         (*********************************************)
         (* parameter 3.7.3 *)
         (*********************************************)
         (
            ParameterName_as8    := 'POL Resistance Min',
            ParameterType_u8     := 0,
            attr1_u              := 0,
            attr2_u              := 3000,
            attr3_u              := 10,
            UnitCode_au8         := 18,
            Multiplier_s16       := 1,
            Divisor_s16          := 1,
            NumberOfDigits_u16   := 0,
            AccesslevelCode_u8   := 179,
            attr4_u              := 2,
            EEPROMAddress_s      := (Page_u8 := 3, IntIndex_u8 := 178)
         ),

         (*********************************************)
         (* parameter 3.7.4 *)
         (*********************************************)
         (
            ParameterName_as8    := 'POL Resistance Max',
            ParameterType_u8     := 0,
            attr1_u              := 0,
            attr2_u              := 3000,
            attr3_u              := 10,
            UnitCode_au8         := 18,
            Multiplier_s16       := 1,
            Divisor_s16          := 1,
            NumberOfDigits_u16   := 0,
            AccesslevelCode_u8   := 179,
            attr4_u              := 52,
            EEPROMAddress_s      := (Page_u8 := 3, IntIndex_u8 := 179)
         ),

         (*********************************************)
         (* parameter 3.7.5 *)
         (*********************************************)
         (
            ParameterName_as8    := 'POL Kp',
            ParameterType_u8     := 0,
            attr1_u              := 0,
            attr2_u              := 2000,
            attr3_u              := 50,
            UnitCode_au8         := 0,
            Multiplier_s16       := 1,
            Divisor_s16          := 1,
            NumberOfDigits_u16   := 0,
            AccesslevelCode_u8   := 179,
            attr4_u              := 250,
            EEPROMAddress_s      := (Page_u8 := 3, IntIndex_u8 := 180)
         ),

         (*********************************************)
         (* parameter 3.7.6 *)
         (*********************************************)
         (
            ParameterName_as8    := 'POL Ki',
            ParameterType_u8     := 0,
            attr1_u              := 0,
            attr2_u              := 500,
            attr3_u              := 50,
            UnitCode_au8         := 0,
            Multiplier_s16       := 1,
            Divisor_s16          := 1,
            NumberOfDigits_u16   := 0,
            AccesslevelCode_u8   := 179,
            attr4_u              := 250,
            EEPROMAddress_s      := (Page_u8 := 3, IntIndex_u8 := 181)
         ),

         (*********************************************)
         (* parameter 3.7.7 *)
         (*********************************************)
         (
         ),

         (*********************************************)
         (* parameter 3.7.8 *)
         (*********************************************)
         (
         )

      ),

      (*********************************************)
      (* parameter group 3.8 - up to 8 parameters can be defined here *)
      (*********************************************)
      (
         GroupName_as8   := 'DOH Configuration',

         Param_as        := 

         (*********************************************)
         (* parameter 3.8.1 *)
         (*********************************************)
         (
            ParameterName_as8    := 'DOH Debounce',
            ParameterType_u8     := 0,
            attr1_u              := 50,
            attr2_u              := 250,
            attr3_u              := 10,
            UnitCode_au8         := 4,
            Multiplier_s16       := 1,
            Divisor_s16          := 1,
            NumberOfDigits_u16   := 0,
            AccesslevelCode_u8   := 179,
            attr4_u              := 200,
            EEPROMAddress_s      := (Page_u8 := 3, IntIndex_u8 := 184)
         ),

         (*********************************************)
         (* parameter 3.8.2 *)
         (*********************************************)
         (
         ),

         (*********************************************)
         (* parameter 3.8.3 *)
         (*********************************************)
         (
            ParameterName_as8    := 'DOH Resistance Min',
            ParameterType_u8     := 0,
            attr1_u              := 0,
            attr2_u              := 3000,
            attr3_u              := 10,
            UnitCode_au8         := 18,
            Multiplier_s16       := 1,
            Divisor_s16          := 1,
            NumberOfDigits_u16   := 0,
            AccesslevelCode_u8   := 179,
            attr4_u              := 6,
            EEPROMAddress_s      := (Page_u8 := 3, IntIndex_u8 := 186)
         ),

         (*********************************************)
         (* parameter 3.8.4 *)
         (*********************************************)
         (
            ParameterName_as8    := 'DOH Resistance Max',
            ParameterType_u8     := 0,
            attr1_u              := 0,
            attr2_u              := 3000,
            attr3_u              := 10,
            UnitCode_au8         := 18,
            Multiplier_s16       := 1,
            Divisor_s16          := 1,
            NumberOfDigits_u16   := 0,
            AccesslevelCode_u8   := 179,
            attr4_u              := 44,
            EEPROMAddress_s      := (Page_u8 := 3, IntIndex_u8 := 187)
         ),

         (*********************************************)
         (* parameter 3.8.5 *)
         (*********************************************)
         (
         ),

         (*********************************************)
         (* parameter 3.8.6 *)
         (*********************************************)
         (
         ),

         (*********************************************)
         (* parameter 3.8.7 *)
         (*********************************************)
         (
         ),

         (*********************************************)
         (* parameter 3.8.8 *)
         (*********************************************)
         (
         )

      )

   ),

   (*********************************************)
   (* parameter menu 4 - up to 8 groups can be defined here *)
   (*********************************************)
   (
   ),

   (*********************************************)
   (* parameter menu 5 - up to 8 groups can be defined here *)
   (*********************************************)
   (
   );


(**)
END_VAR
(*********************************************)
(*  DON'T MAKE ANY CHANGES TO THIS PROGRAM!! *)
(*     FILE WAS AUTOMATICALLY GENERATED!!    *)
(*********************************************)

;
END_PROGRAM

(* POU 05_Basic_Calc/CHARCODE, ST *)
FUNCTION CHARCODE : BYTE
(* Функция получает код (char) для текстового символа *)
VAR_INPUT
	STR : STRING(1);
END_VAR
VAR
	PT : POINTER TO BYTE;
END_VAR
PT := ADR(STR);
CHARCODE := PT^;
END_FUNCTION

(* POU Uds/UdsSrvReadDataByIdServices/UdsGetProcessData, ST *)
PROGRAM UdsGetProcessData

VAR_INPUT
    did: UINT;
END_VAR

VAR
	startIndex: USINT := 1;
	groupNumber: USINT;
	requestedParameter: USINT;

	nonEmptyParametersCount: USINT;
	parameterCounter: USINT;
	numberOfParameters: USINT;
	parameterNameLength : USINT;

	tempCounter: USINT;
END_VAR
did := did - 16#2000;

groupNumber := UINT_TO_BYTE(SHR(did, 4));
groupNumber := groupNumber + 1;
requestedParameter := UINT_TO_BYTE(did) AND 16#0F;
requestedParameter := requestedParameter + 1;
Uds_s.UdsTx.data[1] := 0;

Uds_s.UdsTx.data[1] := Uds_s.UdsTx.data[1] + 1;
Uds_s.UdsTx.data[Uds_s.UdsTx.data[1] + 1 ] := Uds_s.UdsRx.data[2] + 16#40;

numberOfParameters := 8;

IF (LEN(ProcData.ProcessVarGroups_as[groupNumber].GroupName_as8) > 0) THEN
	IF (requestedParameter < 16#08) THEN
		startIndex := requestedParameter;
		numberOfParameters := startIndex;
	END_IF

	FOR parameterCounter := startIndex TO numberOfParameters DO
		parameterNameLength := INT_TO_USINT(LEN(ProcData.ProcessVarGroups_as[groupNumber].GroupName_as8));
		IF (parameterNameLength > 0) THEN
			nonEmptyParametersCount := nonEmptyParametersCount + 1;
		END_IF
	END_FOR

	Uds_s.UdsTx.data[1] := Uds_s.UdsTx.data[1] + 1;
	Uds_s.UdsTx.data[Uds_s.UdsTx.data[1] + 1] := nonEmptyParametersCount;

	FOR parameterCounter := startIndex TO numberOfParameters DO
		parameterNameLength := INT_TO_USINT(LEN(ProcData.ProcessVarGroups_as[groupNumber].GroupName_as8));
		IF (parameternameLength > 0) THEN
			Uds_s.UdsTx.data[1] := Uds_s.UdsTx.data[1] + 1;
			Uds_s.UdsTx.data[Uds_s.UdsTx.data[1] + 1] := parameterCounter - 1;

			IF (ProcData.ProcessVarGroups_as[groupNumber].ProcessVariable_as[parameterCounter].AccesslevelCode_u8 <= Uds_s.activeAccessLevel_u8) THEN
				FOR tempCounter := 1 TO parameterNameLength DO
					Uds_s.UdsTx.data[1] := Uds_s.UdsTx.data[1] + 1;
					Uds_s.UdsTx.data[Uds_s.UdsTx.data[1] + 1] := BYTE_TO_USINT(CHARCODE(MID(ProcData.ProcessVarGroups_as[groupNumber].ProcessVariable_as[parameterCounter].ProcessVarName_as8, 1, tempCounter)));
				END_FOR

				Uds_s.UdsTx.data[1] := Uds_s.UdsTx.data[1] + 1;
				Uds_s.UdsTx.data[Uds_s.UdsTx.data[1] + 1] := 0;

				Uds_s.UdsTx.data[1] := Uds_s.UdsTx.data[1] + 1;
				Uds_s.UdsTx.data[Uds_s.UdsTx.data[1] + 1] := INT_TO_USINT(SHR(ProcData.ProcessVarGroups_as[groupNumber].ProcessVariable_as[parameterCounter].Multiplier_s16, 8));
				Uds_s.UdsTx.data[1] := Uds_s.UdsTx.data[1] + 1;
				Uds_s.UdsTx.data[Uds_s.UdsTx.data[1] + 1] := INT_TO_USINT(ProcData.ProcessVarGroups_as[groupNumber].ProcessVariable_as[parameterCounter].Multiplier_s16);

				Uds_s.UdsTx.data[1] := Uds_s.UdsTx.data[1] + 1;
				Uds_s.UdsTx.data[Uds_s.UdsTx.data[1] + 1] := INT_TO_USINT(SHR(ProcData.ProcessVarGroups_as[groupNumber].ProcessVariable_as[parameterCounter].Divisor_s16, 8));
				Uds_s.UdsTx.data[1] := Uds_s.UdsTx.data[1] + 1;
				Uds_s.UdsTx.data[Uds_s.UdsTx.data[1] + 1] := INT_TO_USINT(ProcData.ProcessVarGroups_as[groupNumber].ProcessVariable_as[parameterCounter].Divisor_s16);

				Uds_s.UdsTx.data[1] := Uds_s.UdsTx.data[1] + 1;
				Uds_s.UdsTx.data[Uds_s.UdsTx.data[1] + 1] := ProcData.ProcessVarGroups_as[groupNumber].ProcessVariable_as[parameterCounter].ProcVarType_u8;

				Uds_s.UdsTx.data[1] := Uds_s.UdsTx.data[1] + 1;
				Uds_s.UdsTx.data[Uds_s.UdsTx.data[1] + 1] := UINT_TO_USINT(SHR(ProcData.ProcessVarGroups_as[groupNumber].ProcessVariable_as[parameterCounter].attr_u, 8));
				Uds_s.UdsTx.data[1] := Uds_s.UdsTx.data[1] + 1;
				Uds_s.UdsTx.data[Uds_s.UdsTx.data[1] + 1] := UINT_TO_USINT(ProcData.ProcessVarGroups_as[groupNumber].ProcessVariable_as[parameterCounter].attr_u);

				Uds_s.UdsTx.data[1] := Uds_s.UdsTx.data[1] + 1;
				Uds_s.UdsTx.data[Uds_s.UdsTx.data[1] + 1] := ProcData.ProcessVarGroups_as[groupNumber].ProcessVariable_as[parameterCounter].UnitCode_au8;

				Uds_s.UdsTx.data[1] := Uds_s.UdsTx.data[1] + 1;
				Uds_s.UdsTx.data[Uds_s.UdsTx.data[1] + 1] := ProcData.ProcessVarGroups_as[groupNumber].ProcessVariable_as[parameterCounter].AccesslevelCode_u8;

				IF (parameterCounter < numberOfParameters - 1 AND LEN(ProcData.ProcessVarGroups_as[groupNumber].ProcessVariable_as[parameterCounter + 1].ProcessVarName_as8) + 12 > (255 - Uds_s.UdsTx.data[1])) THEN
					EXIT;
				END_IF

			ELSE
				Uds_s.UdsTx.data[1] := Uds_s.UdsTx.data[1] + 1;
				Uds_s.UdsTx.data[Uds_s.UdsTx.data[1] + 1] := 0;
			END_IF
		END_IF
	END_FOR

	IF (parameterCounter = numberOfParameters + 1) THEN
		startIndex := 1;
	ELSE
		startIndex := parameterCounter + 1;
	END_IF
END_IF
Uds_s.UdsTx.dataSize := Uds_s.UdsTx.data[1];
END_PROGRAM

(* POU Autocode/ProcData, ST *)
PROGRAM ProcData
(*********************************************)
(*  DON'T MAKE ANY CHANGES TO THIS PROGRAM!! *)
(*     FILE WAS AUTOMATICALLY GENERATED!!    *)
(*********************************************)

VAR
END_VAR
VAR CONSTANT

(**)
(*********************************************)
nrProcMenus_u8          : USINT := 48;

(*********************************************)
(* Process Values Tree *)
(*********************************************)

ProcessVarGroups_as      : ARRAY [1..48] OF ProcessVariableGroup_ts := 

   (*********************************************)
   (* process values group 1 - up to 8 variables can be defined here *)
   (*********************************************)
   (
      GroupName_as8        := 'Group 1',

      ProcessVariable_as   := 

         (*********************************************)
      (* process value 1.1 *)
      (*********************************************)
      (
         ProcessVarName_as8   := 'Param_var',
         ProcVarType_u8       := 0,
         UnitCode_au8         := 1,
         Multiplier_s16       := 1,
         Divisor_s16          := 1,
         attr_u               := 0,
         AccesslevelCode_u8   := 129
      ),
         (*********************************************)
      (* process value 1.2 *)
      (*********************************************)
      (
         ProcessVarName_as8   := 'Param_var',
         ProcVarType_u8       := 0,
         UnitCode_au8         := 1,
         Multiplier_s16       := 1,
         Divisor_s16          := 1,
         attr_u               := 0,
         AccesslevelCode_u8   := 129
      ),
         (*********************************************)
      (* process value 1.3 *)
      (*********************************************)
      (
         ProcessVarName_as8   := 'Param_var',
         ProcVarType_u8       := 0,
         UnitCode_au8         := 1,
         Multiplier_s16       := 1,
         Divisor_s16          := 1,
         attr_u               := 0,
         AccesslevelCode_u8   := 129
      ),
         (*********************************************)
      (* process value 1.4 *)
      (*********************************************)
      (
         ProcessVarName_as8   := 'Param_var',
         ProcVarType_u8       := 0,
         UnitCode_au8         := 1,
         Multiplier_s16       := 1,
         Divisor_s16          := 1,
         attr_u               := 0,
         AccesslevelCode_u8   := 129
      ),
         (*********************************************)
      (* process value 1.5 *)
      (*********************************************)
      (
         ProcessVarName_as8   := 'Param_var',
         ProcVarType_u8       := 0,
         UnitCode_au8         := 0,
         Multiplier_s16       := 1,
         Divisor_s16          := 1,
         attr_u               := 0,
         AccesslevelCode_u8   := 129
      ),
         (*********************************************)
      (* process value 1.6 *)
      (*********************************************)
      (
         ProcessVarName_as8   := 'Param_var',
         ProcVarType_u8       := 0,
         UnitCode_au8         := 0,
         Multiplier_s16       := 1,
         Divisor_s16          := 1,
         attr_u               := 15,
         AccesslevelCode_u8   := 129
      ),
         (*********************************************)
      (* process value 1.7 *)
      (*********************************************)
      (
         ProcessVarName_as8   := 'Param_var',
         ProcVarType_u8       := 0,
         UnitCode_au8         := 0,
         Multiplier_s16       := 1,
         Divisor_s16          := 1,
         attr_u               := 8,
         AccesslevelCode_u8   := 129
      ),
         (*********************************************)
      (* process value 1.8 *)
      (*********************************************)
      (
         ProcessVarName_as8   := 'Param_var',
         ProcVarType_u8       := 0,
         UnitCode_au8         := 0,
         Multiplier_s16       := 1,
         Divisor_s16          := 1,
         attr_u               := 1000,
         AccesslevelCode_u8   := 129
      )
   ),

   (*********************************************)
   (* process values group 2 - up to 8 variables can be defined here *)
   (*********************************************)
   (
      GroupName_as8        := 'Group 2',

      ProcessVariable_as   := 

         (*********************************************)
      (* process value 2.1 *)
      (*********************************************)
      (
         ProcessVarName_as8   := 'Param_var',
         ProcVarType_u8       := 0,
         UnitCode_au8         := 1,
         Multiplier_s16       := 1,
         Divisor_s16          := 1,
         attr_u               := 0,
         AccesslevelCode_u8   := 129
      ),
         (*********************************************)
      (* process value 2.2 *)
      (*********************************************)
      (
         ProcessVarName_as8   := 'Param_var',
         ProcVarType_u8       := 0,
         UnitCode_au8         := 1,
         Multiplier_s16       := 1,
         Divisor_s16          := 1,
         attr_u               := 0,
         AccesslevelCode_u8   := 129
      ),
         (*********************************************)
      (* process value 2.3 *)
      (*********************************************)
      (
         ProcessVarName_as8   := 'Param_var',
         ProcVarType_u8       := 0,
         UnitCode_au8         := 1,
         Multiplier_s16       := 1,
         Divisor_s16          := 1,
         attr_u               := 0,
         AccesslevelCode_u8   := 129
      ),
         (*********************************************)
      (* process value 2.4 *)
      (*********************************************)
      (
         ProcessVarName_as8   := 'Param_var',
         ProcVarType_u8       := 0,
         UnitCode_au8         := 1,
         Multiplier_s16       := 1,
         Divisor_s16          := 1,
         attr_u               := 0,
         AccesslevelCode_u8   := 129
      ),
         (*********************************************)
      (* process value 2.5 *)
      (*********************************************)
      (
         ProcessVarName_as8   := 'Param_var',
         ProcVarType_u8       := 0,
         UnitCode_au8         := 1,
         Multiplier_s16       := 1,
         Divisor_s16          := 1,
         attr_u               := 0,
         AccesslevelCode_u8   := 129
      ),
         (*********************************************)
      (* process value 2.6 *)
      (*********************************************)
      (
         ProcessVarName_as8   := 'Param_var',
         ProcVarType_u8       := 0,
         UnitCode_au8         := 1,
         Multiplier_s16       := 1,
         Divisor_s16          := 1,
         attr_u               := 0,
         AccesslevelCode_u8   := 129
      ),
         (*********************************************)
      (* process value 2.7 *)
      (*********************************************)
      (
         ProcessVarName_as8   := 'Param_var',
         ProcVarType_u8       := 0,
         UnitCode_au8         := 1,
         Multiplier_s16       := 1,
         Divisor_s16          := 1,
         attr_u               := 0,
         AccesslevelCode_u8   := 129
      ),
         (*********************************************)
      (* process value 2.8 *)
      (*********************************************)
      (
         ProcessVarName_as8   := 'Param_var',
         ProcVarType_u8       := 0,
         UnitCode_au8         := 1,
         Multiplier_s16       := 1,
         Divisor_s16          := 1,
         attr_u               := 0,
         AccesslevelCode_u8   := 129
      )
   ),

   (*********************************************)
   (* process values group 3 - up to 8 variables can be defined here *)
   (*********************************************)
   (
      GroupName_as8        := 'Group 3',

      ProcessVariable_as   := 

         (*********************************************)
      (* process value 3.1 *)
      (*********************************************)
      (
         ProcessVarName_as8   := 'Param_var',
         ProcVarType_u8       := 0,
         UnitCode_au8         := 1,
         Multiplier_s16       := 1,
         Divisor_s16          := 1,
         attr_u               := 0,
         AccesslevelCode_u8   := 129
      ),
         (*********************************************)
      (* process value 3.2 *)
      (*********************************************)
      (
         ProcessVarName_as8   := 'Param_var',
         ProcVarType_u8       := 0,
         UnitCode_au8         := 1,
         Multiplier_s16       := 1,
         Divisor_s16          := 1,
         attr_u               := 0,
         AccesslevelCode_u8   := 129
      ),
         (*********************************************)
      (* process value 3.3 *)
      (*********************************************)
      (
         ProcessVarName_as8   := 'Param_var',
         ProcVarType_u8       := 0,
         UnitCode_au8         := 1,
         Multiplier_s16       := 1,
         Divisor_s16          := 1,
         attr_u               := 0,
         AccesslevelCode_u8   := 129
      ),
         (*********************************************)
      (* process value 3.4 *)
      (*********************************************)
      (
         ProcessVarName_as8   := 'Param_var',
         ProcVarType_u8       := 0,
         UnitCode_au8         := 1,
         Multiplier_s16       := 1,
         Divisor_s16          := 1,
         attr_u               := 0,
         AccesslevelCode_u8   := 129
      ),
         (*********************************************)
      (* process value 3.5 *)
      (*********************************************)
      (
         ProcessVarName_as8   := 'Param_var',
         ProcVarType_u8       := 0,
         UnitCode_au8         := 1,
         Multiplier_s16       := 1,
         Divisor_s16          := 1,
         attr_u               := 0,
         AccesslevelCode_u8   := 129
      ),
         (*********************************************)
      (* process value 3.6 *)
      (*********************************************)
      (
         ProcessVarName_as8   := 'Param_var',
         ProcVarType_u8       := 0,
         UnitCode_au8         := 1,
         Multiplier_s16       := 1,
         Divisor_s16          := 1,
         attr_u               := 0,
         AccesslevelCode_u8   := 129
      ),
         (*********************************************)
      (* process value 3.7 *)
      (*********************************************)
      (
         ProcessVarName_as8   := 'Param_var',
         ProcVarType_u8       := 0,
         UnitCode_au8         := 1,
         Multiplier_s16       := 1,
         Divisor_s16          := 1,
         attr_u               := 0,
         AccesslevelCode_u8   := 129
      ),
         (*********************************************)
      (* process value 3.8 *)
      (*********************************************)
      (
         ProcessVarName_as8   := 'Param_var',
         ProcVarType_u8       := 0,
         UnitCode_au8         := 1,
         Multiplier_s16       := 1,
         Divisor_s16          := 1,
         attr_u               := 0,
         AccesslevelCode_u8   := 129
      )
   ),

   (*********************************************)
   (* process values group 4 - up to 8 variables can be defined here *)
   (*********************************************)
   (
      GroupName_as8        := 'Group 4',

      ProcessVariable_as   := 

         (*********************************************)
      (* process value 4.1 *)
      (*********************************************)
      (
         ProcessVarName_as8   := 'Param_var',
         ProcVarType_u8       := 0,
         UnitCode_au8         := 1,
         Multiplier_s16       := 1,
         Divisor_s16          := 1,
         attr_u               := 0,
         AccesslevelCode_u8   := 129
      ),
         (*********************************************)
      (* process value 4.2 *)
      (*********************************************)
      (
         ProcessVarName_as8   := 'Param_var',
         ProcVarType_u8       := 0,
         UnitCode_au8         := 1,
         Multiplier_s16       := 1,
         Divisor_s16          := 1,
         attr_u               := 0,
         AccesslevelCode_u8   := 129
      ),
         (*********************************************)
      (* process value 4.3 *)
      (*********************************************)
      (
         ProcessVarName_as8   := 'Param_var',
         ProcVarType_u8       := 0,
         UnitCode_au8         := 1,
         Multiplier_s16       := 1,
         Divisor_s16          := 1,
         attr_u               := 0,
         AccesslevelCode_u8   := 129
      ),
         (*********************************************)
      (* process value 4.4 *)
      (*********************************************)
      (
         ProcessVarName_as8   := 'Param_var',
         ProcVarType_u8       := 0,
         UnitCode_au8         := 1,
         Multiplier_s16       := 1,
         Divisor_s16          := 1,
         attr_u               := 0,
         AccesslevelCode_u8   := 129
      ),
         (*********************************************)
      (* process value 4.5 *)
      (*********************************************)
      (
         ProcessVarName_as8   := 'Param_var',
         ProcVarType_u8       := 0,
         UnitCode_au8         := 1,
         Multiplier_s16       := 1,
         Divisor_s16          := 1,
         attr_u               := 0,
         AccesslevelCode_u8   := 129
      ),
         (*********************************************)
      (* process value 4.6 *)
      (*********************************************)
      (
         ProcessVarName_as8   := 'Param_var',
         ProcVarType_u8       := 0,
         UnitCode_au8         := 1,
         Multiplier_s16       := 1,
         Divisor_s16          := 1,
         attr_u               := 0,
         AccesslevelCode_u8   := 129
      ),
         (*********************************************)
      (* process value 4.7 *)
      (*********************************************)
      (
         ProcessVarName_as8   := 'Param_var',
         ProcVarType_u8       := 0,
         UnitCode_au8         := 1,
         Multiplier_s16       := 1,
         Divisor_s16          := 1,
         attr_u               := 0,
         AccesslevelCode_u8   := 129
      ),
         (*********************************************)
      (* process value 4.8 *)
      (*********************************************)
      (
      )
   ),

   (*********************************************)
   (* process values group 5 - up to 8 variables can be defined here *)
   (*********************************************)
   (
      GroupName_as8        := 'Group 5',

      ProcessVariable_as   := 

         (*********************************************)
      (* process value 5.1 *)
      (*********************************************)
      (
         ProcessVarName_as8   := 'Param_var',
         ProcVarType_u8       := 0,
         UnitCode_au8         := 1,
         Multiplier_s16       := 1,
         Divisor_s16          := 1,
         attr_u               := 0,
         AccesslevelCode_u8   := 129
      ),
         (*********************************************)
      (* process value 5.2 *)
      (*********************************************)
      (
         ProcessVarName_as8   := 'Param_var',
         ProcVarType_u8       := 0,
         UnitCode_au8         := 1,
         Multiplier_s16       := 1,
         Divisor_s16          := 1,
         attr_u               := 0,
         AccesslevelCode_u8   := 129
      ),
         (*********************************************)
      (* process value 5.3 *)
      (*********************************************)
      (
         ProcessVarName_as8   := 'Param_var',
         ProcVarType_u8       := 0,
         UnitCode_au8         := 1,
         Multiplier_s16       := 1,
         Divisor_s16          := 1,
         attr_u               := 0,
         AccesslevelCode_u8   := 129
      ),
         (*********************************************)
      (* process value 5.4 *)
      (*********************************************)
      (
         ProcessVarName_as8   := 'Param_var',
         ProcVarType_u8       := 0,
         UnitCode_au8         := 1,
         Multiplier_s16       := 1,
         Divisor_s16          := 1,
         attr_u               := 0,
         AccesslevelCode_u8   := 129
      ),
         (*********************************************)
      (* process value 5.5 *)
      (*********************************************)
      (
         ProcessVarName_as8   := 'Param_var',
         ProcVarType_u8       := 0,
         UnitCode_au8         := 1,
         Multiplier_s16       := 1,
         Divisor_s16          := 1,
         attr_u               := 0,
         AccesslevelCode_u8   := 129
      ),
         (*********************************************)
      (* process value 5.6 *)
      (*********************************************)
      (
         ProcessVarName_as8   := 'Param_var',
         ProcVarType_u8       := 0,
         UnitCode_au8         := 1,
         Multiplier_s16       := 1,
         Divisor_s16          := 1,
         attr_u               := 0,
         AccesslevelCode_u8   := 129
      ),
         (*********************************************)
      (* process value 5.7 *)
      (*********************************************)
      (
      ),
         (*********************************************)
      (* process value 5.8 *)
      (*********************************************)
      (
      )
   ),

   (*********************************************)
   (* process values group 6 - up to 8 variables can be defined here *)
   (*********************************************)
   (


   ),

   (*********************************************)
   (* process values group 7 - up to 8 variables can be defined here *)
   (*********************************************)
   (


   ),

   (*********************************************)
   (* process values group 8 - up to 8 variables can be defined here *)
   (*********************************************)
   (


   ),

   (*********************************************)
   (* process values group 9 - up to 8 variables can be defined here *)
   (*********************************************)
   (


   ),

   (*********************************************)
   (* process values group 10 - up to 8 variables can be defined here *)
   (*********************************************)
   (


   ),

   (*********************************************)
   (* process values group 11 - up to 8 variables can be defined here *)
   (*********************************************)
   (


   ),

   (*********************************************)
   (* process values group 12 - up to 8 variables can be defined here *)
   (*********************************************)
   (


   ),

   (*********************************************)
   (* process values group 13 - up to 8 variables can be defined here *)
   (*********************************************)
   (


   ),

   (*********************************************)
   (* process values group 14 - up to 8 variables can be defined here *)
   (*********************************************)
   (


   ),

   (*********************************************)
   (* process values group 15 - up to 8 variables can be defined here *)
   (*********************************************)
   (


   ),

   (*********************************************)
   (* process values group 16 - up to 8 variables can be defined here *)
   (*********************************************)
   (


   ),

   (*********************************************)
   (* process values group 17 - up to 8 variables can be defined here *)
   (*********************************************)
   (


   ),

   (*********************************************)
   (* process values group 18 - up to 8 variables can be defined here *)
   (*********************************************)
   (


   ),

   (*********************************************)
   (* process values group 19 - up to 8 variables can be defined here *)
   (*********************************************)
   (


   ),

   (*********************************************)
   (* process values group 20 - up to 8 variables can be defined here *)
   (*********************************************)
   (


   ),

   (*********************************************)
   (* process values group 21 - up to 8 variables can be defined here *)
   (*********************************************)
   (


   ),

   (*********************************************)
   (* process values group 22 - up to 8 variables can be defined here *)
   (*********************************************)
   (


   ),

   (*********************************************)
   (* process values group 23 - up to 8 variables can be defined here *)
   (*********************************************)
   (


   ),

   (*********************************************)
   (* process values group 24 - up to 8 variables can be defined here *)
   (*********************************************)
   (


   ),

   (*********************************************)
   (* process values group 25 - up to 8 variables can be defined here *)
   (*********************************************)
   (


   ),

   (*********************************************)
   (* process values group 26 - up to 8 variables can be defined here *)
   (*********************************************)
   (


   ),

   (*********************************************)
   (* process values group 27 - up to 8 variables can be defined here *)
   (*********************************************)
   (


   ),

   (*********************************************)
   (* process values group 28 - up to 8 variables can be defined here *)
   (*********************************************)
   (


   ),

   (*********************************************)
   (* process values group 29 - up to 8 variables can be defined here *)
   (*********************************************)
   (


   ),

   (*********************************************)
   (* process values group 30 - up to 8 variables can be defined here *)
   (*********************************************)
   (


   ),

   (*********************************************)
   (* process values group 31 - up to 8 variables can be defined here *)
   (*********************************************)
   (


   ),

   (*********************************************)
   (* process values group 32 - up to 8 variables can be defined here *)
   (*********************************************)
   (


   ),

   (*********************************************)
   (* process values group 33 - up to 8 variables can be defined here *)
   (*********************************************)
   (


   ),

   (*********************************************)
   (* process values group 34 - up to 8 variables can be defined here *)
   (*********************************************)
   (


   ),

   (*********************************************)
   (* process values group 35 - up to 8 variables can be defined here *)
   (*********************************************)
   (


   ),

   (*********************************************)
   (* process values group 36 - up to 8 variables can be defined here *)
   (*********************************************)
   (


   ),

   (*********************************************)
   (* process values group 37 - up to 8 variables can be defined here *)
   (*********************************************)
   (


   ),

   (*********************************************)
   (* process values group 38 - up to 8 variables can be defined here *)
   (*********************************************)
   (


   ),

   (*********************************************)
   (* process values group 39 - up to 8 variables can be defined here *)
   (*********************************************)
   (


   ),

   (*********************************************)
   (* process values group 40 - up to 8 variables can be defined here *)
   (*********************************************)
   (


   ),

   (*********************************************)
   (* process values group 41 - up to 8 variables can be defined here *)
   (*********************************************)
   (


   ),

   (*********************************************)
   (* process values group 42 - up to 8 variables can be defined here *)
   (*********************************************)
   (


   ),

   (*********************************************)
   (* process values group 43 - up to 8 variables can be defined here *)
   (*********************************************)
   (


   ),

   (*********************************************)
   (* process values group 44 - up to 8 variables can be defined here *)
   (*********************************************)
   (


   ),

   (*********************************************)
   (* process values group 45 - up to 8 variables can be defined here *)
   (*********************************************)
   (


   ),

   (*********************************************)
   (* process values group 46 - up to 8 variables can be defined here *)
   (*********************************************)
   (


   ),

   (*********************************************)
   (* process values group 47 - up to 8 variables can be defined here *)
   (*********************************************)
   (


   ),

   (*********************************************)
   (* process values group 48 - up to 8 variables can be defined here *)
   (*********************************************)
   (


   );


(**)
END_VAR
(*********************************************)
(*  DON'T MAKE ANY CHANGES TO THIS PROGRAM!! *)
(*     FILE WAS AUTOMATICALLY GENERATED!!    *)
(*********************************************)

;
END_PROGRAM

(* POU Uds/UdsSrvReadDataByIdServices/UdsGetParameterMenuNames, ST *)
PROGRAM UdsGetParameterMenuNames
VAR
	startIndex: USINT := 1;
	menuCounter: USINT;
	menuNameLength: USINT;

	nonEmptyMenuNamesCounter: USINT;
	tempCounter: USINT;
END_VAR
Uds_s.UdsTx.data[1] := 0;

Uds_s.UdsTx.data[1] := Uds_s.UdsTx.data[1] + 1;
Uds_s.UdsTx.data[Uds_s.UdsTx.data[1] + 1 ] := Uds_s.UdsRx.data[2] + 16#40;

FOR menuCounter := startIndex TO PrmData.nrPrmMenus_u8 DO
	menuNameLength := INT_TO_USINT(LEN(PrmData.ParameterMenus_as[menuCounter].MenuName_as8));
	IF (menuNameLength > 0) THEN
		nonEmptyMenuNamesCounter := nonEmptyMenuNamesCounter + 1;
	END_IF
END_FOR

Uds_s.UdsTx.data[1] := Uds_s.UdsTx.data[1] + 1;
Uds_s.UdsTx.data[Uds_s.UdsTx.data[1] + 1 ] := nonEmptyMenuNamesCounter;

FOR menuCounter := startIndex TO PrmData.nrPrmMenus_u8 DO
	menuNameLength := INT_TO_USINT(LEN(PrmData.ParameterMenus_as[menuCounter].MenuName_as8));
	IF (menuNameLength > 0) THEN
		Uds_s.UdsTx.data[1] := Uds_s.UdsTx.data[1] + 1;
		Uds_s.UdsTx.data[Uds_s.UdsTx.data[1] + 1] := menuCounter - 1;

		FOR tempCounter := 1 TO menuNameLength DO
			Uds_s.UdsTx.data[1] := Uds_s.UdsTx.data[1] + 1;
			Uds_s.UdsTx.data[Uds_s.UdsTx.data[1] + 1] := BYTE_TO_USINT(CHARCODE(MID(PrmData.ParameterMenus_as[menuCounter].MenuName_as8, 1, tempCounter)));
		END_FOR

		Uds_s.UdsTx.data[1] := Uds_s.UdsTx.data[1] + 1;
		Uds_s.UdsTx.data[Uds_s.UdsTx.data[1] + 1] := 0;

		IF (menuCounter < PrmData.nrPrmMenus_u8 - 1 AND LEN(PrmData.ParameterMenus_as[menuCounter + 1].MenuName_as8) + 3 > 255 - Uds_s.UdsTx.data[1]) THEN
			EXIT;
		END_IF
	END_IF
END_FOR
IF (menuCounter = PrmData.nrPrmMenus_u8 + 1) THEN
	startIndex := 1;
ELSE
	startIndex := menuCounter + 1;
END_IF
Uds_s.UdsTx.dataSize := Uds_s.UdsTx.data[1];
END_PROGRAM

(* POU Uds/UdsSrvReadDataByIdServices/UdsGetParameterSubMenuNames, ST *)
PROGRAM UdsGetParameterSubMenuNames

VAR_INPUT
    did: UINT;
END_VAR

VAR
	startIndex: USINT := 1;

	menuNumber: USINT;
	numberOfSubmenuNames: USINT := 8;
	subMenuCounter: USINT;
	nonEmptySubMenuNamesCounter: USINT;
	subMenuNameLength: USINT;

	tempCounter: USINT;
END_VAR
did := did - 16#2201;
menuNumber := UINT_TO_USINT(did);

Uds_s.UdsTx.data[1] := 0;
Uds_s.UdsTx.data[1] := Uds_s.UdsTx.data[1] + 1;
Uds_s.UdsTx.data[Uds_s.UdsTx.data[1] + 1 ] := Uds_s.UdsRx.data[2] + 16#40;

IF (LEN(PrmData.ParameterMenus_as[menuNumber].MenuName_as8) > 0) THEN
	FOR subMenuCounter := startIndex TO numberOfSubmenuNames DO
		subMenuNameLength := INT_TO_USINT(LEN(PrmData.ParameterMenus_as[menuNumber].ParameterGroup_as[subMenuCounter].GroupName_as8));
		IF (subMenuNameLength > 0) THEN
			nonEmptySubMenuNamesCounter := nonEmptySubMenuNamesCounter + 1;
		END_IF
	END_FOR

	Uds_s.UdsTx.data[1] := Uds_s.UdsTx.data[1] + 1;
	Uds_s.UdsTx.data[Uds_s.UdsTx.data[1] + 1 ] := nonEmptySubMenuNamesCounter;

	FOR subMenuCounter := startIndex TO numberOfSubmenuNames DO
		subMenuNameLength := INT_TO_USINT(LEN(PrmData.ParameterMenus_as[menuNumber].ParameterGroup_as[subMenuCounter].GroupName_as8));
		IF (subMenuNameLength > 0) THEN
			Uds_s.UdsTx.data[1] := Uds_s.UdsTx.data[1] + 1;
			Uds_s.UdsTx.data[Uds_s.UdsTx.data[1] + 1 ] := subMenuCounter;

			FOR tempCounter := 1 TO subMenuNameLength DO
				Uds_s.UdsTx.data[1] := Uds_s.UdsTx.data[1] + 1;
				Uds_s.UdsTx.data[Uds_s.UdsTx.data[1] + 1] := BYTE_TO_USINT(CHARCODE(MID(PrmData.ParameterMenus_as[menuNumber].ParameterGroup_as[subMenuCounter].GroupName_as8, 1, tempCounter)));
			END_FOR

			Uds_s.UdsTx.data[1] := Uds_s.UdsTx.data[1] + 1;
			Uds_s.UdsTx.data[Uds_s.UdsTx.data[1] + 1 ] := 0;

			IF (subMenuCounter < numberOfSubmenuNames - 1 AND LEN(PrmData.ParameterMenus_as[menuNumber].ParameterGroup_as[subMenuCounter + 1].GroupName_as8) + 3 > 255 - Uds_s.UdsTx.data[1]) THEN
				EXIT;
			END_IF
		END_IF
	END_FOR
	IF (subMenuCounter = numberOfSubmenuNames + 1) THEN
		startIndex := 1;
	ELSE
		startIndex := subMenuCounter + 1;
	END_IF
END_IF
Uds_s.UdsTx.dataSize := Uds_s.UdsTx.data[1];
END_PROGRAM

(* POU Uds/UdsSrvReadDataByIdServices/UdsGetProcessGroupNames, ST *)
PROGRAM UdsGetProcessGroupNames
VAR
    groupCounter : USINT;
    startIndex : USINT := 1;
    tempCounter : USINT;
    groupNameLength : USINT;
	nonEmptyGroupNamesCounter: USINT;
END_VAR
Uds_s.UdsTx.data[1] := Uds_s.UdsTx.data[1] + 1;
Uds_s.UdsTx.data[Uds_s.UdsTx.data[1] + 1 ] := Uds_s.UdsRx.data[2] + 16#40;

FOR groupCounter := startIndex TO ProcData.nrProcMenus_u8 DO
	groupNameLength := INT_TO_USINT(LEN(ProcData.ProcessVarGroups_as[groupCounter].GroupName_as8));
	IF (groupNameLength > 0) THEN
		nonEmptyGroupNamesCounter := nonEmptyGroupNamesCounter + 1;
	END_IF
END_FOR

Uds_s.UdsTx.data[1] := Uds_s.UdsTx.data[1] + 1;
Uds_s.UdsTx.data[Uds_s.UdsTx.data[1] + 1 ] := nonEmptyGroupNamesCounter;

FOR groupCounter := startIndex TO ProcData.nrProcMenus_u8 DO
    groupNameLength := INT_TO_USINT(LEN(ProcData.ProcessVarGroups_as[groupCounter].GroupName_as8));
    IF groupNameLength > 0 THEN
        Uds_s.UdsTx.data[1] := Uds_s.UdsTx.data[1] + 1;
        Uds_s.UdsTx.data[Uds_s.UdsTx.data[1] + 1] := groupCounter - 1;


        FOR tempCounter := 1 TO groupNameLength DO
            Uds_s.UdsTx.data[1] := Uds_s.UdsTx.data[1] + 1;
            Uds_s.UdsTx.data[Uds_s.UdsTx.data[1] + 1] := BYTE_TO_USINT(CHARCODE(MID(ProcData.ProcessVarGroups_as[groupCounter].GroupName_as8, 1, tempCounter)));
        END_FOR

        Uds_s.UdsTx.data[1] := Uds_s.UdsTx.data[1] + 1;
        Uds_s.UdsTx.data[Uds_s.UdsTx.data[1] + 1] := 0;
        IF (groupCounter < ProcData.nrProcMenus_u8 - 1 AND LEN(ProcData.ProcessVarGroups_as[groupCounter].GroupName_as8) + 3 > 255 - Uds_s.UdsTx.data[1]) THEN
            EXIT;
        END_IF
    END_IF
END_FOR
IF (groupCounter = ProcData.nrProcMenus_u8 + 1) THEN
    startIndex := 1;
ELSE
    startIndex := groupCounter + 1;
END_IF
Uds_s.UdsTx.dataSize := Uds_s.UdsTx.data[1];
END_PROGRAM

(* POU Uds/UdsSrvReadDataByIdServices/UdsGetUnitCodes, ST *)
PROGRAM UdsGetUnitCodes
VAR
    startIndex_u16 : USINT := 1;
    unitCodeCounter : USINT;
    tempCounter : USINT;
    unitCodeLength : USINT;
END_VAR
Uds_s.UdsTx.data[1] := 0;

Uds_s.UdsTx.data[1] := Uds_s.UdsTx.data[1] + 1;
Uds_s.UdsTx.data[Uds_s.UdsTx.data[1] + 1 ] := Uds_s.UdsRx.data[2] + 16#40;

Uds_s.UdsTx.data[1] := Uds_s.UdsTx.data[1] + 1;
Uds_s.UdsTx.data[Uds_s.UdsTx.data[1] + 1 ] := UnitCodes.nrUnitCodes_u8;

FOR unitCodeCounter := startIndex_u16 TO UnitCodes.nrUnitCodes_u8 DO
    Uds_s.UdsTx.data[1] := Uds_s.UdsTx.data[1] + 1;
    Uds_s.UdsTx.data[Uds_s.UdsTx.data[1] + 1] := unitCodeCounter - 1;
    unitCodeLength := INT_TO_USINT(LEN(UnitCodes.UnitCodes_cau8[unitCodeCounter]));
    FOR tempCounter := 1 TO unitCodeLength DO
        Uds_s.UdsTx.data[1] := Uds_s.UdsTx.data[1] + 1;
        Uds_s.UdsTx.data[Uds_s.UdsTx.data[1] + 1] := BYTE_TO_USINT(CHARCODE(MID(UnitCodes.UnitCodes_cau8[unitCodeCounter], 1, tempCounter)));
    END_FOR
    Uds_s.UdsTx.data[1] := Uds_s.UdsTx.data[1] + 1;
    Uds_s.UdsTx.data[Uds_s.UdsTx.data[1] + 1] := 0;

    IF (unitCodeCounter < UnitCodes.nrUnitCodes_u8 AND LEN(UnitCodes.UnitCodes_cau8[unitCodeCounter + 1]) + 3 > (255 - Uds_s.UdsTx.data[1])) THEN
        EXIT;
    END_IF
END_FOR

IF (unitCodeCounter = UnitCodes.nrUnitCodes_u8) THEN
    startIndex_u16 := 1;
ELSE
    startIndex_u16 := unitCodeCounter + 1;
END_IF
Uds_s.UdsTx.dataSize := Uds_s.UdsTx.data[1];
END_PROGRAM

(* POU Autocode/UnitCodes, ST *)
PROGRAM UnitCodes
(*********************************************)
(*  DON'T MAKE ANY CHANGES TO THIS PROGRAM!! *)
(*     FILE WAS AUTOMATICALLY GENERATED!!    *)
(*********************************************)

VAR
END_VAR
VAR CONSTANT

(**)
(*********************************************)
nrUnitCodes_u8      : USINT := 18;

(*********************************************)
(* Unit Codes Array *)

UnitCodes_cau8      : ARRAY [1..18] OF STRING(8) := 
   '%',
   'rpm',
   'hrs',
   'ms',
   'ccm',
   'mA',
   'bar',
   'mbar',
   'Deg C',
   'min',
   's',
   'km/h',
   'Nm',
   'deg °',
   '% / mA',
   '% / mV',
   'uA / mV',
   'Ohm';


(**)
END_VAR
(*********************************************)
(*  DON'T MAKE ANY CHANGES TO THIS PROGRAM!! *)
(*     FILE WAS AUTOMATICALLY GENERATED!!    *)
(*********************************************)

;
END_PROGRAM

(* POU Uds/UdsSrvReadDataByIdServices/UdsGetListDescriptions, ST *)
PROGRAM UdsGetListDescriptions
VAR
	listEntriesCounter: UINT;
	numberOfEntries: UINT;
	nonEmptyListDescriptionsCounter: UINT;
	listEntryLength: USINT;

	startIndex: UINT := 1;
	tempCounter: USINT;
END_VAR
Uds_s.UdsTx.data[1] := 0;

Uds_s.UdsTx.data[1] := Uds_s.UdsTx.data[1] + 1;
Uds_s.UdsTx.data[Uds_s.UdsTx.data[1] + 1 ] := Uds_s.UdsRx.data[2] + 16#40;

numberOfEntries := Lists.nrLists_u8 * 10;

FOR listEntriesCounter := startIndex TO numberOfEntries DO
	listEntryLength := INT_TO_USINT(LEN(Lists.ParaLists_as[listEntriesCounter / 10 + 1][listEntriesCounter MOD 10]));
	IF (listEntryLength > 0) THEN
		nonEmptyListDescriptionsCounter := nonEmptyListDescriptionsCounter + 1;
	END_IF
END_FOR

Uds_s.UdsTx.data[1] := Uds_s.UdsTx.data[1] + 1;
Uds_s.UdsTx.data[Uds_s.UdsTx.data[1] + 1 ] := UINT_TO_USINT(SHR(nonEmptyListDescriptionsCounter, 8));

Uds_s.UdsTx.data[1] := Uds_s.UdsTx.data[1] + 1;
Uds_s.UdsTx.data[Uds_s.UdsTx.data[1] + 1 ] := UINT_TO_USINT(nonEmptyListDescriptionsCounter);

Uds_s.UdsTx.data[1] := Uds_s.UdsTx.data[1] + 1;
Uds_s.UdsTx.data[Uds_s.UdsTx.data[1] + 1 ] := 10;

FOR listEntriesCounter := startIndex TO numberOfEntries DO
	listEntryLength := INT_TO_USINT(LEN(Lists.ParaLists_as[listEntriesCounter / 10 + 1][listEntriesCounter MOD 10]));
	IF (listEntryLength > 0) THEN
		Uds_s.UdsTx.data[1] := Uds_s.UdsTx.data[1] + 1;
		Uds_s.UdsTx.data[Uds_s.UdsTx.data[1] + 1 ] := UINT_TO_USINT(SHR(listEntriesCounter, 8));

		Uds_s.UdsTx.data[1] := Uds_s.UdsTx.data[1] + 1;
		Uds_s.UdsTx.data[Uds_s.UdsTx.data[1] + 1 ] := UINT_TO_USINT(listEntriesCounter);

		FOR tempCounter := 1 TO listEntryLength DO
			Uds_s.UdsTx.data[1] := Uds_s.UdsTx.data[1] + 1;
			Uds_s.UdsTx.data[Uds_s.UdsTx.data[1] + 1] := BYTE_TO_USINT(CHARCODE(MID(Lists.ParaLists_as[listEntriesCounter / 10 + 1][listEntriesCounter MOD 10], 1, tempCounter)));
		END_FOR

		Uds_s.UdsTx.data[1] := Uds_s.UdsTx.data[1] + 1;
		Uds_s.UdsTx.data[Uds_s.UdsTx.data[1] + 1] := 0;

		IF (listEntriesCounter <  numberOfEntries - 1 AND LEN(Lists.ParaLists_as[(listEntriesCounter + 1) / 10 + 1][(listEntriesCounter + 1) MOD 10]) > (255 - Uds_s.UdsTx.data[1])) THEN
			EXIT;
		END_IF
	END_IF
END_FOR

IF (listEntriesCounter = numberOfEntries + 1) THEN
	startIndex := 1;
ELSE
	startIndex := listEntriesCounter + 1;
END_IF

Uds_s.UdsTx.dataSize := Uds_s.UdsTx.data[1];
END_PROGRAM

(* POU Autocode/Lists, ST *)
PROGRAM Lists
(*********************************************)
(*  DON'T MAKE ANY CHANGES TO THIS PROGRAM!! *)
(*     FILE WAS AUTOMATICALLY GENERATED!!    *)
(*********************************************)

VAR
END_VAR
VAR CONSTANT

(**)
(*********************************************)
nrLists_u8      : USINT := 4;

(*********************************************)
(* Lists Tree*)

ParaLists_as      : ARRAY [1..4] OF ARRAY[1..10] OF STRING(32) := 
      'Not Active',
      'Active',
      '',
      '',
      '',
      '',
      '',
      '',
      '',
      '',
      'PWM',
      'PWM Current control',
      '',
      '',
      '',
      '',
      '',
      '',
      '',
      '',
      'PWM',
      'AOV',
      '',
      '',
      '',
      '',
      '',
      '',
      '',
      '',
      'AOC',
      'AOV',
      '',
      '',
      '',
      '',
      '',
      '',
      '',
      ''
;

(**)
END_VAR
(*********************************************)
(*  DON'T MAKE ANY CHANGES TO THIS PROGRAM!! *)
(*     FILE WAS AUTOMATICALLY GENERATED!!    *)
(*********************************************)

;
END_PROGRAM

(* POU Uds/UdsSrvReadDataByIdServices/UdsGetErrors, ST *)
PROGRAM UdsGetErrors
VAR_INPUT
    errorType: USINT;
END_VAR
VAR
    numErr : USINT;
    errorData : ARRAY[1..50] OF ErrorData_ts;
    errorCounter : USINT;
    startIndex : USINT := 1;
    tempCounter : USINT;
    errorListCounter : USINT;
    errorsEnum : applError_e;
END_VAR
Uds_s.UdsTx.data[1] := Uds_s.UdsTx.data[1] + 1;
Uds_s.UdsTx.data[Uds_s.UdsTx.data[1] + 1 ] := Uds_s.UdsRx.data[2] + 16#40;

IF (errorType = 0) THEN
    numErr := UINT_TO_USINT(sys_getSavedErrors(ADR(errorData[1]), 0, 50));
ELSIF (errorType = 1) THEN
    numErr := UINT_TO_USINT(sys_getActiveErrors(ADR(errorData[1]), 0, 50));
(*ELSE
    (*7F*)*)
END_IF

FOR errorCounter := startIndex TO numErr DO
    IF errorData[errorCounter].Code_u16 = 0 THEN
        EXIT;
    END_IF
    Uds_s.UdsTx.data[1] := Uds_s.UdsTx.data[1] + 1;
    Uds_s.UdsTx.data[Uds_s.UdsTx.data[1] + 1] := UINT_TO_USINT(SHR(errorData[errorCounter].Code_u16, 8));
    Uds_s.UdsTx.data[1] := Uds_s.UdsTx.data[1] + 1;
    Uds_s.UdsTx.data[Uds_s.UdsTx.data[1] + 1] := UINT_TO_USINT(errorData[errorCounter].Code_u16);
    Uds_s.UdsTx.data[1] := Uds_s.UdsTx.data[1] + 1;
    Uds_s.UdsTx.data[Uds_s.UdsTx.data[1] + 1] := errorData[errorCounter].Param_u8;
    Uds_s.UdsTx.data[1] := Uds_s.UdsTx.data[1] + 1;
    Uds_s.UdsTx.data[Uds_s.UdsTx.data[1] + 1] := errorData[errorCounter].Occurrence_u8;
    Uds_s.UdsTx.data[1] := Uds_s.UdsTx.data[1] + 1;
    Uds_s.UdsTx.data[Uds_s.UdsTx.data[1] + 1] := UDINT_TO_USINT(SHR(errorData[errorCounter].Timestamp_u32, 24));
    Uds_s.UdsTx.data[1] := Uds_s.UdsTx.data[1] + 1;
    Uds_s.UdsTx.data[Uds_s.UdsTx.data[1] + 1] := UDINT_TO_USINT(SHR(errorData[errorCounter].Timestamp_u32, 16));
    Uds_s.UdsTx.data[1] := Uds_s.UdsTx.data[1] + 1;
    Uds_s.UdsTx.data[Uds_s.UdsTx.data[1] + 1] := UDINT_TO_USINT(SHR(errorData[errorCounter].Timestamp_u32, 8));
    Uds_s.UdsTx.data[1] := Uds_s.UdsTx.data[1] + 1;
    Uds_s.UdsTx.data[Uds_s.UdsTx.data[1] + 1] := UDINT_TO_USINT(errorData[errorCounter].Timestamp_u32);

    FOR errorListCounter := 0 TO ErrorsList.nrErrors_u8 DO
        IF ErrorsList.ApplError_as[errorListCounter].Code_u16 = errorData[errorCounter].Code_u16 THEN
            FOR tempCounter := 0 TO INT_TO_USINT(LEN(ErrorsList.ApplError_as[errorListCounter].Description_as8)) DO
                Uds_s.UdsTx.data[1] := Uds_s.UdsTx.data[1] + 1;
                Uds_s.UdsTx.data[Uds_s.UdsTx.data[1] + 1] := BYTE_TO_USINT(CHARCODE(MID(ErrorsList.ApplError_as[errorListCounter].Description_as8, 1, tempCounter)));
            END_FOR
        END_IF
    END_FOR
END_FOR
IF (errorCounter = numErr + 1) THEN
    startIndex := 1;
ELSE
    startIndex := errorCounter + 1;
END_IF
Uds_s.UdsTx.dataSize := Uds_s.UdsTx.data[1];
END_PROGRAM

(* POU Autocode/ErrorsList, ST *)
PROGRAM ErrorsList
(*********************************************)
(*  DON'T MAKE ANY CHANGES TO THIS ENUMS!!   *)
(*     FILE WAS AUTOMATICALLY GENERATED!!    *)
(*********************************************)
VAR
END_VAR
VAR CONSTANT

(**)
(*********************************************)

(* Errors Tree *)
(*********************************************)
nrErrors_u8          : USINT := 21;

(*********************************************)
ApplError_as      : ARRAY [1..21] OF ApplErrorNew_ts := 

   (
      Code_u16 := 16#8000,
      Description_as8 := 'FIRST_CODE'
   ),
   (
      Code_u16 := 16#8001,
      Description_as8 := 'CAN_DIAG'
   ),
   (
      Code_u16 := 16#8036,
      Description_as8 := 'PWRON_SUPPLY_VB_LOW'
   ),
   (
      Code_u16 := 16#8037,
      Description_as8 := 'PWRON_SUPPLY_VSS'
   ),
   (
      Code_u16 := 16#8038,
      Description_as8 := 'PWRON_HWMONITOR_1'
   ),
   (
      Code_u16 := 16#8039,
      Description_as8 := 'PWRON_STARTCONDITION_1'
   ),
   (
      Code_u16 := 16#8040,
      Description_as8 := 'PWRON_ENGINE_SPEED'
   ),
   (
      Code_u16 := 16#8041,
      Description_as8 := 'PWRON_HWMONITOR_2'
   ),
   (
      Code_u16 := 16#8042,
      Description_as8 := 'PWRON_STARTCONDITION_2'
   ),
   (
      Code_u16 := 16#8043,
      Description_as8 := 'PWRON_SAFOUT_CABLE_BRAKE'
   ),
   (
      Code_u16 := 16#8044,
      Description_as8 := 'PWRON_SAFOUT_SHORT_CIRCUIT'
   ),
   (
      Code_u16 := 16#8045,
      Description_as8 := 'PWRON_POWERSWITCH_1'
   ),
   (
      Code_u16 := 16#8046,
      Description_as8 := 'PWRON_POWERSUPPLY'
   ),
   (
      Code_u16 := 16#8047,
      Description_as8 := 'PWRON_POWERSWITCH_2'
   ),
   (
      Code_u16 := 16#8048,
      Description_as8 := 'PWRON_REVERSE_POWER'
   ),
   (
      Code_u16 := 16#8049,
      Description_as8 := 'PWRON_EMERGENCY_STOP'
   ),
   (
      Code_u16 := 16#8031,
      Description_as8 := 'SUPPLY_VB_HIGH'
   ),
   (
      Code_u16 := 16#8032,
      Description_as8 := 'SUPPLY_VB_LOW'
   ),
   (
      Code_u16 := 16#8033,
      Description_as8 := 'SUPPLY_VSS1'
   ),
   (
      Code_u16 := 16#8034,
      Description_as8 := 'SUPPLY_VSS2'
   ),
   (
      Code_u16 := 16#8099,
      Description_as8 := 'LAST_CODE'
   )
(**)
;
END_VAR
(*********************************************)
(*  DON'T MAKE ANY CHANGES TO THIS PROGRAM!! *)
(*     FILE WAS AUTOMATICALLY GENERATED!!    *)
(*********************************************)

;
END_PROGRAM

(* POU Uds/UdsSrvReadDataByIdServices/UdsDidAcsPrm, ST *)
PROGRAM UdsDidAcsPrm
VAR_INPUT
	did: UINT;
   flgWrDid: USINT;
END_VAR
VAR
	menuNumber:USINT;
	subMenuNumber: USINT;
	parameterNumber: USINT;
	rawVal: UINT;
END_VAR
(* TODO
Запись: проверка на другие размеры передаваемого значения (1 байт, размер = 4)
*)
menuNumber := UINT_TO_BYTE(SHR(did, 7)) AND 16#3F;
menuNumber := menuNumber + 1;
subMenuNumber := UINT_TO_BYTE(SHR(did, 4)) AND 16#07;
subMenuNumber := subMenuNumber + 1;
parameterNumber := UINT_TO_BYTE(did) AND 16#0F;
parameterNumber := parameterNumber + 1;

IF (menuNumber <= PrmData.nrPrmMenus_u8) THEN

Uds_s.UdsTx.data[1] := 0;

Uds_s.UdsTx.data[1] := Uds_s.UdsTx.data[1] + 1;
Uds_s.UdsTx.data[Uds_s.UdsTx.data[1] + 1 ] := Uds_s.UdsRx.data[2] + 16#40;

IF (flgWrDid = 0) THEN (*read access*)
	rawVal := ree_getValue(PrmData.ParameterMenus_as[menuNumber].ParameterGroup_as[subMenuNumber].Param_as[parameterNumber].EEPROMAddress_s.Page_u8,
									PrmData.ParameterMenus_as[menuNumber].ParameterGroup_as[subMenuNumber].Param_as[parameterNumber].EEPROMAddress_s.IntIndex_u8);
	Uds_s.UdsTx.data[1] := Uds_s.UdsTx.data[1] + 1;
	Uds_s.UdsTx.data[Uds_s.UdsTx.data[1] + 1 ] := UINT_TO_USINT(SHR(did, 8));
	Uds_s.UdsTx.data[1] := Uds_s.UdsTx.data[1] + 1;
	Uds_s.UdsTx.data[Uds_s.UdsTx.data[1] + 1 ] := UINT_TO_USINT(did);

ELSE (*write access*)
	IF Uds_s.UdsRx.dataSize = 5 THEN (*1 - sid; 2,3 - did; 4,5 - value*)
		rawVal := USINT_TO_UINT(SHL(Uds_s.UdsRx.data[4], 8));
		rawVal := rawVal + Uds_s.UdsRx.data[5];
		IF (rawVal > PrmData.ParameterMenus_as[menuNumber].ParameterGroup_as[subMenuNumber].Param_as[parameterNumber].attr1_u AND
				rawVal < PrmData.ParameterMenus_as[menuNumber].ParameterGroup_as[subMenuNumber].Param_as[parameterNumber].attr2_u) THEN
			ree_setValue(PrmData.ParameterMenus_as[menuNumber].ParameterGroup_as[subMenuNumber].Param_as[parameterNumber].EEPROMAddress_s.Page_u8,
								PrmData.ParameterMenus_as[menuNumber].ParameterGroup_as[subMenuNumber].Param_as[parameterNumber].EEPROMAddress_s.IntIndex_u8,
								rawVal);
		END_IF
	END_IF
END_IF
Uds_s.UdsTx.dataSize := Uds_s.UdsTx.data[1];

END_IF
END_PROGRAM

(* POU Uds/UdsSrvReadDataByIdServices/UdsDidAcsProcVal, ST *)
PROGRAM UdsDidAcsProcVal
VAR_INPUT
	did : UINT;
END_VAR
VAR
END_VAR
;
END_PROGRAM

(* POU Uds/UdsSrvWriteDataById, ST *)
PROGRAM UdsSrvWriteDataById
VAR
	didus : UINT;
END_VAR
IF (Uds_s.UdsRx.dataSize > 0 AND Uds_s.UdsRx.data[1] > 0) THEN
	didus := Uds_s.UdsRx.data[3];
	didus := SHL(didus, 8);
	didus := didus + Uds_s.UdsRx.data[4];

	UdsDidAcsPrm(did := didus, flgWrDid := 1);
END_IF
END_PROGRAM

(* POU Uds/UdsSrvTesterPresent, ST *)
PROGRAM UdsSrvTesterPresent
VAR

END_VAR
IF(Uds_s.UdsRx.dataSize = 2) THEN
	Uds_s.UdsTx.data[1] := 0;
	
	Uds_s.UdsTx.data[1] := Uds_s.UdsTx.data[1] + 1;
	Uds_s.UdsTx.data[Uds_s.UdsTx.data[1] + 1 ] := Uds_s.UdsRx.data[2] + 16#40;

	Uds_s.UdsTx.data[1] := Uds_s.UdsTx.data[1] + 1;
	Uds_s.UdsTx.data[Uds_s.UdsTx.data[1] + 1 ] := 16#00;
	
	Uds_s.UdsTx.dataSize := Uds_s.UdsTx.data[1];
END_IF
END_PROGRAM

(* POU Autocode/Callback_update_appl_param, ST *)
(*************************************************************************************
BRIEF: read the whole parameters from the EEPROM
*************************************************************************************
 (c) Copyright by BOSCH REXROTH AG, all rights reserved 
*************************************************************************************
VERSION INFORMATION
	V1.0 	Vitaly Lewitan, DC-MA/SMC
- Call Autocode parameter assignment programm
- Update (or Init) function block parameters

REVISION HISTORY:
	V1.0 	Vitaly Lewitan, DC-MA/SMC
 - 23/03-2012 Initial Version
**************************************************************************************)
PROGRAM Callback_update_appl_param

VAR
   eep:  ARRAY [0..1280] OF INT;
END_VAR
Callback_diag_getPara();
(* Get_Aggregate_param(); *)
END_PROGRAM

(* POU Autocode/Callback_diag_getPara, ST *)
PROGRAM Callback_diag_getPara
VAR
   eep:  ARRAY [0..1280] OF INT;
END_VAR
(*********************************************)
(*  DON'T MAKE ANY CHANGES TO THIS PROGRAM!! *)
(*     FILE WAS AUTOMATICALLY GENERATED!!    *)
(*********************************************)

(* get EEPROM pages 0..4 *)
ree_getArray( PAGE0, 0, ADR(eep[0]),    256 );
ree_getArray( PAGE1, 0, ADR(eep[256]),  256 );
ree_getArray( PAGE2, 0, ADR(eep[512]),  256 );
ree_getArray( PAGE3, 0, ADR(eep[768]),  256 );
ree_getArray( PAGE4, 0, ADR(eep[1024]), 256 );


(* Menu 1 *)

(* Basic *)
para_s.number_1_1_1_s16 := eep[EEP_number_1_1_1_e];
para_s.Input_to_Output_Mode_s16 := eep[EEP_Input_to_Output_Mode_e];
para_s.test_par_new_s16 := eep[EEP_test_par_new_e];
para_s.test_params_s16 := eep[EEP_test_params_e];
para_s.test_par2_s16 := eep[EEP_test_par2_e];

(* Test Type *)
para_s.Trimming_type_s16 := eep[EEP_Trimming_type_e];
para_s.Analog_type_s16 := eep[EEP_Analog_type_e];
para_s.Curve_Type_s16 := eep[EEP_Curve_Type_e];
para_s.Function_Type_s16 := eep[EEP_Function_Type_e];
para_s.Percent_Type_s16 := eep[EEP_Percent_Type_e];
para_s.Ramp_Type_s16 := eep[EEP_Ramp_Type_e];
para_s.Switch_Type_s16 := eep[EEP_Switch_Type_e];
para_s.List_Type_s16 := eep[EEP_List_Type_e];

(* Test Number *)
para_s.number_1_3_1_s16 := eep[EEP_number_1_3_1_e];
para_s.number_1_3_2_s16 := eep[EEP_number_1_3_2_e];
para_s.number_1_3_3_s16 := eep[EEP_number_1_3_3_e];
para_s.number_1_3_4_s16 := eep[EEP_number_1_3_4_e];
para_s.number_1_3_5_s16 := eep[EEP_number_1_3_5_e];
para_s.number_1_3_6_s16 := eep[EEP_number_1_3_6_e];
para_s.number_1_3_7_s16 := eep[EEP_number_1_3_7_e];
para_s.number_1_3_8_s16 := eep[EEP_number_1_3_8_e];


(* Menu 2 *)

(* Output Cfg 1-8 *)
para_s.Out_Cfg_01_s16 := eep[EEP_Out_Cfg_01_e];
para_s.Out_Cfg_02_s16 := eep[EEP_Out_Cfg_02_e];
para_s.Out_Cfg_03_s16 := eep[EEP_Out_Cfg_03_e];
para_s.Out_Cfg_04_s16 := eep[EEP_Out_Cfg_04_e];
para_s.Out_Cfg_05_s16 := eep[EEP_Out_Cfg_05_e];
para_s.Out_Cfg_06_s16 := eep[EEP_Out_Cfg_06_e];
para_s.Out_Cfg_07_s16 := eep[EEP_Out_Cfg_07_e];
para_s.Out_Cfg_08_s16 := eep[EEP_Out_Cfg_08_e];

(* Output Cfg 9-16 *)
para_s.Out_Cfg_09_s16 := eep[EEP_Out_Cfg_09_e];
para_s.Out_Cfg_10_s16 := eep[EEP_Out_Cfg_10_e];
para_s.Out_Cfg_11_s16 := eep[EEP_Out_Cfg_11_e];
para_s.Out_Cfg_12_s16 := eep[EEP_Out_Cfg_12_e];
para_s.Out_Cfg_13_s16 := eep[EEP_Out_Cfg_13_e];
para_s.Out_Cfg_14_s16 := eep[EEP_Out_Cfg_14_e];
para_s.Out_Cfg_15_s16 := eep[EEP_Out_Cfg_15_e];
para_s.Out_Cfg_16_s16 := eep[EEP_Out_Cfg_16_e];

(* Output Cfg 17-24 *)
para_s.Out_Cfg_17_s16 := eep[EEP_Out_Cfg_17_e];
para_s.Out_Cfg_18_s16 := eep[EEP_Out_Cfg_18_e];
para_s.Out_Cfg_19_s16 := eep[EEP_Out_Cfg_19_e];
para_s.Out_Cfg_20_s16 := eep[EEP_Out_Cfg_20_e];
para_s.Out_Cfg_21_s16 := eep[EEP_Out_Cfg_21_e];
para_s.Out_Cfg_22_s16 := eep[EEP_Out_Cfg_22_e];
para_s.Out_Cfg_23_s16 := eep[EEP_Out_Cfg_23_e];
para_s.Out_Cfg_24_s16 := eep[EEP_Out_Cfg_24_e];

(* Output Cfg 25-32 *)
para_s.Out_Cfg_25_s16 := eep[EEP_Out_Cfg_25_e];
para_s.Out_Cfg_26_s16 := eep[EEP_Out_Cfg_26_e];
para_s.Out_Cfg_27_s16 := eep[EEP_Out_Cfg_27_e];
para_s.Out_Cfg_28_s16 := eep[EEP_Out_Cfg_28_e];
para_s.Out_Cfg_29_s16 := eep[EEP_Out_Cfg_29_e];
para_s.Out_Cfg_30_s16 := eep[EEP_Out_Cfg_30_e];
para_s.Out_Cfg_31_s16 := eep[EEP_Out_Cfg_31_e];
para_s.Out_Cfg_32_s16 := eep[EEP_Out_Cfg_32_e];

(* Output Cfg 33-40 *)
para_s.Out_Cfg_33_s16 := eep[EEP_Out_Cfg_33_e];
para_s.Out_Cfg_34_s16 := eep[EEP_Out_Cfg_34_e];
para_s.Out_Cfg_35_s16 := eep[EEP_Out_Cfg_35_e];
para_s.Out_Cfg_36_s16 := eep[EEP_Out_Cfg_36_e];
para_s.Out_Cfg_37_s16 := eep[EEP_Out_Cfg_37_e];
para_s.Out_Cfg_38_s16 := eep[EEP_Out_Cfg_38_e];
para_s.Out_Cfg_39_s16 := eep[EEP_Out_Cfg_39_e];
para_s.Out_Cfg_40_s16 := eep[EEP_Out_Cfg_40_e];

(* Output Cfg 41-47 *)
para_s.Out_Cfg_41_s16 := eep[EEP_Out_Cfg_41_e];
para_s.Out_Cfg_42_s16 := eep[EEP_Out_Cfg_42_e];
para_s.Out_Cfg_43_s16 := eep[EEP_Out_Cfg_43_e];
para_s.Out_Cfg_44_s16 := eep[EEP_Out_Cfg_44_e];
para_s.Out_Cfg_45_s16 := eep[EEP_Out_Cfg_45_e];
para_s.Out_Cfg_46_s16 := eep[EEP_Out_Cfg_46_e];
para_s.Out_Cfg_47_s16 := eep[EEP_Out_Cfg_47_e];

(* AOV Configuration *)
para_s.AOV_Debounce_s16 := eep[EEP_AOV_Debounce_e];
para_s.AOV_Freq_s16 := eep[EEP_AOV_Freq_e];
para_s.AOV_Res_Min_s16 := eep[EEP_AOV_Res_Min_e];
para_s.AOV_Res_Max_s16 := eep[EEP_AOV_Res_Max_e];
para_s.AOV_Kp_s16 := eep[EEP_AOV_Kp_e];
para_s.AOV_Ki_s16 := eep[EEP_AOV_Ki_e];

(* AOC Configuration *)
para_s.AOC_Debounce_s16 := eep[EEP_AOC_Debounce_e];
para_s.AOC_Freq_s16 := eep[EEP_AOC_Freq_e];
para_s.AOC_Res_Min_s16 := eep[EEP_AOC_Res_Min_e];
para_s.AOC_Res_Max_s16 := eep[EEP_AOC_Res_Max_e];
para_s.AOC_Kp_s16 := eep[EEP_AOC_Kp_e];
para_s.AOC_Ki_s16 := eep[EEP_AOC_Ki_e];


(* Menu 3 *)

(* Output Value 1-8 *)
para_s.Out_Val_01_s16 := eep[EEP_Out_Val_01_e];
para_s.Out_Val_02_s16 := eep[EEP_Out_Val_02_e];
para_s.Out_Val_03_s16 := eep[EEP_Out_Val_03_e];
para_s.Out_Val_04_s16 := eep[EEP_Out_Val_04_e];
para_s.Out_Val_05_s16 := eep[EEP_Out_Val_05_e];
para_s.Out_Val_06_s16 := eep[EEP_Out_Val_06_e];
para_s.Out_Val_07_s16 := eep[EEP_Out_Val_07_e];
para_s.Out_Val_08_s16 := eep[EEP_Out_Val_08_e];

(* Output Value 9-16 *)
para_s.Out_Val_09_s16 := eep[EEP_Out_Val_09_e];
para_s.Out_Val_10_s16 := eep[EEP_Out_Val_10_e];
para_s.Out_Val_11_s16 := eep[EEP_Out_Val_11_e];
para_s.Out_Val_12_s16 := eep[EEP_Out_Val_12_e];
para_s.Out_Val_13_s16 := eep[EEP_Out_Val_13_e];
para_s.Out_Val_14_s16 := eep[EEP_Out_Val_14_e];
para_s.Out_Val_15_s16 := eep[EEP_Out_Val_15_e];
para_s.Out_Val_16_s16 := eep[EEP_Out_Val_16_e];

(* Output Value 17-36 *)
para_s.Out_Val_17_s16 := eep[EEP_Out_Val_17_e];
para_s.Out_Val_18_s16 := eep[EEP_Out_Val_18_e];
para_s.Out_Val_33_s16 := eep[EEP_Out_Val_33_e];
para_s.Out_Val_34_s16 := eep[EEP_Out_Val_34_e];
para_s.Out_Val_35_s16 := eep[EEP_Out_Val_35_e];
para_s.Out_Val_36_s16 := eep[EEP_Out_Val_36_e];

(* Output Value 37-44 *)
para_s.Out_Val_37_s16 := eep[EEP_Out_Val_37_e];
para_s.Out_Val_38_s16 := eep[EEP_Out_Val_38_e];
para_s.Out_Val_39_s16 := eep[EEP_Out_Val_39_e];
para_s.Out_Val_40_s16 := eep[EEP_Out_Val_40_e];
para_s.Out_Val_41_s16 := eep[EEP_Out_Val_41_e];
para_s.Out_Val_42_s16 := eep[EEP_Out_Val_42_e];
para_s.Out_Val_43_s16 := eep[EEP_Out_Val_43_e];
para_s.Out_Val_44_s16 := eep[EEP_Out_Val_44_e];

(* Output Value 45-47 *)
para_s.Out_Val_45_s16 := eep[EEP_Out_Val_45_e];
para_s.Out_Val_46_s16 := eep[EEP_Out_Val_46_e];
para_s.Out_Val_47_s16 := eep[EEP_Out_Val_47_e];

(* POH Configuration *)
para_s.POH_Debounce_s16 := eep[EEP_POH_Debounce_e];
para_s.POH_Res_Min_s16 := eep[EEP_POH_Res_Min_e];
para_s.POH_Res_Max_s16 := eep[EEP_POH_Res_Max_e];
para_s.POH_Kp_s16 := eep[EEP_POH_Kp_e];
para_s.POH_Ki_s16 := eep[EEP_POH_Ki_e];

(* POL Configuration *)
para_s.POL_Debounce_s16 := eep[EEP_POL_Debounce_e];
para_s.POL_Res_Min_s16 := eep[EEP_POL_Res_Min_e];
para_s.POL_Res_Max_s16 := eep[EEP_POL_Res_Max_e];
para_s.POL_Kp_s16 := eep[EEP_POL_Kp_e];
para_s.POL_Ki_s16 := eep[EEP_POL_Ki_e];

(* DOH Configuration *)
para_s.DOH_Debounce_s16 := eep[EEP_DOH_Debounce_e];
para_s.DOH_Res_Min_s16 := eep[EEP_DOH_Res_Min_e];
para_s.DOH_Res_Max_s16 := eep[EEP_DOH_Res_Max_e];
END_PROGRAM

(* POU SwInfo, ST *)
PROGRAM SwInfo
VAR

	SwInfo_lenString_DU32	: INT := 255;
	Eep_sizePage_16bit_D		: INT := 256;

	SwInfo_strSep_DAS8		: STRING := ' |-| \n\r';
	SwInfo_dataString_as8	: STRING(255);

	idx_u16						: INT := 1;

	flgCompRes_u8				: BOOL := FALSE;

	SwInfo_dataEepromRd_as16 : ARRAY[1..256] OF INT := 0;
	SwInfo_dataEepromWr_as16 : ARRAY[1..256] OF INT := 0;

	Ecu_nrEepPageEcuInfo_D	: INT := 32;
END_VAR
(* copy constant SW Name string to target *)
SwInfo_dataString_as8 := 'Software Git Commit Hash: ';
SwInfo_dataString_as8 := CONCAT(SwInfo_dataString_as8, SW_Version.SW_Git_Hash_as8);
SwInfo_dataString_as8 := CONCAT(SwInfo_dataString_as8, ';');


(* switch byte order in string *)
(* Switch byte order of characters in string to prepare string for display in BODAS service *)
FOR idx_u16 := 1 TO SwInfo_lenString_DU32 BY 1 DO
	IF (idx_u16 MOD 2 = 0) THEN
		(* odd byte position *)
		SwInfo_dataEepromWr_as16[idx_u16/2] := WORD_TO_INT(INT_TO_WORD(SwInfo_dataEepromWr_as16[idx_u16/2]) OR (BYTE_TO_WORD(CHARCODE(MID(SwInfo_dataString_as8, 1, idx_u16)))  AND 16#00FF));
	ELSE
		(* even byte position *)
		SwInfo_dataEepromWr_as16[idx_u16/2 + 1] :=  WORD_TO_INT(SHL(BYTE_TO_WORD(CHARCODE(MID(SwInfo_dataString_as8, 1, idx_u16))),8) AND 16#FF00);
	END_IF
END_FOR

(* read current content of EEPROM RAM mirror page containing ECU information *)
ree_getArray(Ecu_nrEepPageEcuInfo_D, 0, ADR(SwInfo_dataEepromRd_as16[1]), Eep_sizePage_16bit_D);

(* create index for array comparison *)
idx_u16 := 1;

(* create flag holding array comparison result *)
flgCompRes_u8 := FALSE;
(* -------------------------------------------------------------------------------------------- *)

(* compare actual content with intended content *)
WHILE ((idx_u16 < Eep_sizePage_16bit_D) AND (NOT flgCompRes_u8)) DO
	IF (SwInfo_dataEepromRd_as16[idx_u16] <> SwInfo_dataEepromWr_as16[idx_u16]) THEN
		flgCompRes_u8 := TRUE;
	END_IF
	idx_u16 := idx_u16 + 1;
END_WHILE

IF (flgCompRes_u8) THEN
	ee_saveArray(Ecu_nrEepPageEcuInfo_D, 0, ADR(SwInfo_dataEepromWr_as16[1]), Eep_sizePage_16bit_D);
END_IF
END_PROGRAM

(* POU 10_Inputs/General Parameters/Get_System_Info, ST *)
PROGRAM Get_System_Info
VAR
	stSupplyVP1_b8			: BOOL;	(*state of the supply VP1*)
	stSupplyVP2_b8			: BOOL;	(*state of the supply VP2*)

	tiSysRunTime_s32		: DINT;	(*duration of the task*)
	etaSysTaskLoad_s16	: INT;	(*load of the main task*)

	stSysEMCY_b8			: BOOL; (*State of the emergency switch*)
	stSysINH_b8				: BOOL;	(*State of INH (pin228)*)

	PCB_temp_s16			: INT;  (*temperature of the RC*)

	error_u16				: UINT;	(* ECU info error *)
	EcuInfo_s				: EcuInfo_ts;
   errors_u16				: ARRAY [1..19] OF UINT;
   BufferAPPL_au8			: ARRAY [1..32] OF USINT;
   BufferSB_au8			: ARRAY [1..6] OF USINT;
   BufferCB_au8			: ARRAY [1..6] OF USINT;
   BufferAPI_au8			: ARRAY [1..1024] OF USINT;
   BufferAPs_au8			: ARRAY [1..19] OF ARRAY [1..16] OF USINT;
   copiedBytes_u16		: ARRAY [1..19] OF UINT;
END_VAR
(********************************************************************************************)
(******************** Checkt:INH / EMCY state  **********************************************)
(********************************************************************************************)
(*check the state OF 'INH': excepted value: OFF*)
stSysINH_b8		:= USINT_TO_BOOL(sys_getINH());
stSysEMCY_b8	:= emcy_getStatus( );
(******************************************************************************)
(******************** Read Supply Voltage  ************************************)
(******************************************************************************)
(* check VP switches *)
stSupplyVP1_b8		:= sys_getVP( VP_1 );			(* State of the supply VP1 *)
stSupplyVP2_b8		:= sys_getVP( VP_2 );			(* State of the supply VP2 *)
(******************************************************************************)
(******************** Read Task data  *****************************************)
(******************************************************************************)
tiSysRunTime_s32 		:= sys_getTaskRunTime( PLC_PRG.MAIN_Task_Handle_u8, PTIME_AVERAGE_INCL );
etaSysTaskLoad_s16 	:= sys_getTaskLoad(PTIME_AVERAGE_INCL);
(******************************************************************************)
(******************** Reads the PCB (Printed circuit board) temperature in °C**)
(******************************************************************************)
PCB_temp_s16 := sys_getHwTemp(AIT_HW_1);

(* Get information of the electronic circuit unit (ECU) *)
error_u16 := sys_getEcuInfo(ADR(EcuInfo_s));

(*
errors_u16[1] 	:= sys_getVersion(VERSION_SW_PART_APPL_DU8 					, ADR(BufferAPPL_au8[1]), 	32,	ADR(copiedBytes_u16[1]));
errors_u16[2] 	:= sys_getVersion(VERSION_SW_PART_SB_DU8						, ADR(BufferSB_au8[1]), 	6, 	ADR(copiedBytes_u16[2]));
errors_u16[3] 	:= sys_getVersion(VERSION_SW_PART_CB_DU8						, ADR(BufferCB_au8[1]), 	6, 	ADR(copiedBytes_u16[3]));
errors_u16[4] 	:= sys_getVersion(VERSION_SW_PART_API_ALL_DU8 				, ADR(BufferAPI_au8[1]), 	1024,	ADR(copiedBytes_u16[4]));
errors_u16[5] 	:= sys_getVersion(VERSION_SW_PART_API_BASIC_DU8 			, ADR(BufferAPs_au8[5]), 	16,	ADR(copiedBytes_u16[5]));
errors_u16[6] 	:= sys_getVersion(VERSION_SW_PART_API_SRC_RC_BASIC_DU8 	, ADR(BufferAPs_au8[6]), 	16,	ADR(copiedBytes_u16[6]));
errors_u16[7] 	:= sys_getVersion(VERSION_SW_PART_API_EEPROM_DU8 			, ADR(BufferAPs_au8[7]), 	16,	ADR(copiedBytes_u16[7]));
errors_u16[8] 	:= sys_getVersion(VERSION_SW_PART_API_DIAG_DU8 				, ADR(BufferAPs_au8[8]), 	16,	ADR(copiedBytes_u16[8]));
errors_u16[9] 	:= sys_getVersion(VERSION_SW_PART_API_INEXT_DU8 			, ADR(BufferAPs_au8[9]), 	16,	ADR(copiedBytes_u16[9]));
errors_u16[10] := sys_getVersion(VERSION_SW_PART_API_STM_DU8	 			, ADR(BufferAPs_au8[10]), 	16,	ADR(copiedBytes_u16[10]));
errors_u16[11] := sys_getVersion(VERSION_SW_PART_API_CANOPEN_DU8 			, ADR(BufferAPs_au8[11]), 	16,	ADR(copiedBytes_u16[11]));
errors_u16[12] := sys_getVersion(VERSION_SW_PART_API_J1939_DU8 			, ADR(BufferAPs_au8[12]), 	16,	ADR(copiedBytes_u16[12]));
errors_u16[13] := sys_getVersion(VERSION_SW_PART_API_RTS_DU8	 			, ADR(BufferAPs_au8[13]), 	16,	ADR(copiedBytes_u16[13]));
errors_u16[14] := sys_getVersion(VERSION_SW_PART_API_CANOPEN_RCE_DU8		, ADR(BufferAPs_au8[14]), 	16,	ADR(copiedBytes_u16[14]));
errors_u16[15] := sys_getVersion(VERSION_SW_PART_API_UDS_DU8	 			, ADR(BufferAPs_au8[15]), 	16,	ADR(copiedBytes_u16[15]));
errors_u16[16] := sys_getVersion(VERSION_SW_PART_API_OUTEXT_DU8 			, ADR(BufferAPs_au8[16]), 	16,	ADR(copiedBytes_u16[16]));
errors_u16[17] := sys_getVersion(VERSION_SW_PART_API_ACOM_DU8	 			, ADR(BufferAPs_au8[17]), 	16,	ADR(copiedBytes_u16[17]));
errors_u16[18]	:= sys_getVersion(VERSION_SW_PART_API_RTM_DU8	 			, ADR(BufferAPs_au8[18]), 	16,	ADR(copiedBytes_u16[18]));
errors_u16[19]	:= sys_getVersion(VERSION_SW_PART_API_CCP_DU8	 			, ADR(BufferAPs_au8[19]), 	16,	ADR(copiedBytes_u16[19]));
*)
END_PROGRAM

(* POU 30_Outputs/out_Control, ST *)
PROGRAM out_Control
VAR
	out_19_state_b8	: BOOL;	(* Состояние выхода out_19 *)
	out_19_status_s	: out_ts;	(* Статус выхода out_19 *)
	out_19_on_b8		: BOOL;

	out_Brakes_status_s	: out_ts;	(* Статус выхода out_19 *)
	out_Brakes_on_b8		: BOOL;
END_VAR
VAR CONSTANT
	DOH_DUTYCYCLE_ON		: UINT	:= 10000;	(* Скважность, при которой дискретный выход активирован *)
END_VAR
IF para_s.Input_to_Output_Mode_s16 = DEACTIVATED THEN


	out_POH();
	out_DOH();
	out_AOV();
	out_POL();

IF PLC_PRG.EcuInfo_s.HwType_u16 <> PLC_PRG.HW_Type_RC12_10_30_u16 THEN
	out_getStatusxt(IO_Chnl.DOH_BRAKES, ADR(out_Brakes_status_s));
	out_Brakes_on_b8		:= out_Brakes_status_s.out_po_s.dc_u16 = DOH_DUTYCYCLE_ON;

	out(IO_Chnl.DOH_FLASHING_BEACON,	BOOL_TO_INT(out_Brakes_on_b8));							(* Выход маяка *)
END_IF

ELSE


;
END_IF
END_PROGRAM
ACTION out_AOV:
IF para_s.Out_Cfg_33_s16 = PWM_MODE THEN
	out (	OUT_33_POH,	para_s.Out_Val_33_s16);
ELSIF para_s.Out_Cfg_33_s16 = AOV_MODE THEN
	out (	OUT_33_AOV,	para_s.Out_Val_33_s16);
END_IF

IF para_s.Out_Cfg_34_s16 = PWM_MODE THEN
	out (	OUT_34_POH,	para_s.Out_Val_34_s16);
ELSIF para_s.Out_Cfg_34_s16 = AOV_MODE THEN
	out (	OUT_34_AOV,	para_s.Out_Val_34_s16);
END_IF

IF para_s.Out_Cfg_35_s16 = PWM_MODE THEN
	out (	OUT_35_POH,	para_s.Out_Val_35_s16);
ELSIF para_s.Out_Cfg_35_s16 = AOV_MODE THEN
	out (	OUT_35_AOV,	para_s.Out_Val_35_s16);
END_IF

IF para_s.Out_Cfg_36_s16 = PWM_MODE THEN
	out (	OUT_36_POH,	para_s.Out_Val_36_s16);
ELSIF para_s.Out_Cfg_36_s16 = AOV_MODE THEN
	out (	OUT_36_AOV,	para_s.Out_Val_36_s16);
END_IF

IF para_s.Out_Cfg_47_s16 = AOC_MODE THEN
	out (	OUT_47_AOC,	para_s.Out_Val_47_s16);
ELSIF para_s.Out_Cfg_47_s16 = AOV_MODE THEN
	out (	OUT_47_AOV,	para_s.Out_Val_47_s16);
END_IF
END_ACTION
ACTION out_DOH:
out(OUT_19_DOH, para_s.Out_Cfg_19_s16);
out(OUT_20_DOH, para_s.Out_Cfg_20_s16);
out(OUT_21_DOH, para_s.Out_Cfg_21_s16);
out(OUT_22_DOH, para_s.Out_Cfg_22_s16);
out(OUT_23_DOH, para_s.Out_Cfg_23_s16);
out(OUT_24_DOH, para_s.Out_Cfg_24_s16);
out(OUT_25_DOH, para_s.Out_Cfg_25_s16);
out(OUT_26_DOH, para_s.Out_Cfg_26_s16);
out(OUT_27_DOH, para_s.Out_Cfg_27_s16);
out(OUT_28_DOH, para_s.Out_Cfg_28_s16);
out(OUT_29_DOH, para_s.Out_Cfg_29_s16);
out(OUT_30_DOH, para_s.Out_Cfg_30_s16);
out(OUT_31_DOH, para_s.Out_Cfg_31_s16);
out(OUT_32_DOH, para_s.Out_Cfg_32_s16);
END_ACTION
ACTION out_POH:
(* Proportional output high side PWM *)

IF para_s.Out_Cfg_01_s16 = PWM_MODE THEN
	out (	OUT_1_POH,	para_s.Out_Val_01_s16);
ELSIF para_s.Out_Cfg_01_s16 = PWM_CURRENT_MODE THEN
	out (	OUT_1_POH_CL,	para_s.Out_Val_01_s16);
END_IF

IF para_s.Out_Cfg_02_s16 = PWM_MODE THEN
	out (	OUT_2_POH,	para_s.Out_Val_02_s16);
ELSIF para_s.Out_Cfg_01_s16 = PWM_CURRENT_MODE THEN
	out (	OUT_2_POH_CL,	para_s.Out_Val_02_s16);
END_IF

IF para_s.Out_Cfg_03_s16 = PWM_MODE THEN
	out (	OUT_3_POH,	para_s.Out_Val_03_s16);
ELSIF para_s.Out_Cfg_03_s16 = PWM_CURRENT_MODE THEN
	out (	OUT_3_POH_CL,	para_s.Out_Val_03_s16);
END_IF

IF para_s.Out_Cfg_04_s16 = PWM_MODE THEN
	out (	OUT_4_POH,	para_s.Out_Val_04_s16);
ELSIF para_s.Out_Cfg_04_s16 = PWM_CURRENT_MODE THEN
	out (	OUT_4_POH_CL,	para_s.Out_Val_04_s16);
END_IF

IF para_s.Out_Cfg_05_s16 = PWM_MODE THEN
	out (	OUT_5_POH,	para_s.Out_Val_05_s16);
ELSIF para_s.Out_Cfg_05_s16 = PWM_CURRENT_MODE THEN
	out (	OUT_5_POH_CL,	para_s.Out_Val_05_s16);
END_IF

IF para_s.Out_Cfg_06_s16 = PWM_MODE THEN
	out (	OUT_6_POH,	para_s.Out_Val_06_s16);
ELSIF para_s.Out_Cfg_06_s16 = PWM_CURRENT_MODE THEN
	out (	OUT_6_POH_CL,	para_s.Out_Val_06_s16);
END_IF

IF para_s.Out_Cfg_07_s16 = PWM_MODE THEN
	out (	OUT_7_POH,	para_s.Out_Val_07_s16);
ELSIF para_s.Out_Cfg_07_s16 = PWM_CURRENT_MODE THEN
	out (	OUT_7_POH_CL,	para_s.Out_Val_07_s16);
END_IF

IF para_s.Out_Cfg_08_s16 = PWM_MODE THEN
	out (	OUT_8_POH,	para_s.Out_Val_08_s16);
ELSIF para_s.Out_Cfg_08_s16 = PWM_CURRENT_MODE THEN
	out (	OUT_8_POH_CL,	para_s.Out_Val_08_s16);
END_IF

IF para_s.Out_Cfg_09_s16 = PWM_MODE THEN
	out (	OUT_9_POH,	para_s.Out_Val_09_s16);
ELSIF para_s.Out_Cfg_09_s16 = PWM_CURRENT_MODE THEN
	out (	OUT_9_POH_CL,	para_s.Out_Val_09_s16);
END_IF

IF para_s.Out_Cfg_10_s16 = PWM_MODE THEN
	out (	OUT_10_POH,	para_s.Out_Val_10_s16);
ELSIF para_s.Out_Cfg_10_s16 = PWM_CURRENT_MODE THEN
	out (	OUT_10_POH_CL,	para_s.Out_Val_10_s16);
END_IF

IF para_s.Out_Cfg_11_s16 = PWM_MODE THEN
	out (	OUT_11_POH,	para_s.Out_Val_11_s16);
ELSIF para_s.Out_Cfg_11_s16 = PWM_CURRENT_MODE THEN
	out (	OUT_11_POH_CL,	para_s.Out_Val_11_s16);
END_IF

IF para_s.Out_Cfg_12_s16 = PWM_MODE THEN
	out (	OUT_12_POH,	para_s.Out_Val_12_s16);
ELSIF para_s.Out_Cfg_12_s16 = PWM_CURRENT_MODE THEN
	out (	OUT_12_POH_CL,	para_s.Out_Val_12_s16);
END_IF

IF para_s.Out_Cfg_13_s16 = PWM_MODE THEN
	out (	OUT_13_POH,	para_s.Out_Val_13_s16);
ELSIF para_s.Out_Cfg_13_s16 = PWM_CURRENT_MODE THEN
	out (	OUT_13_POH_CL,	para_s.Out_Val_13_s16);
END_IF

IF para_s.Out_Cfg_14_s16 = PWM_MODE THEN
	out (	OUT_14_POH,	para_s.Out_Val_14_s16);
ELSIF para_s.Out_Cfg_14_s16 = PWM_CURRENT_MODE THEN
	out (	OUT_14_POH_CL,	para_s.Out_Val_14_s16);
END_IF

IF para_s.Out_Cfg_15_s16 = PWM_MODE THEN
	out (	OUT_15_POH,	para_s.Out_Val_15_s16);
ELSIF para_s.Out_Cfg_15_s16 = PWM_CURRENT_MODE THEN
	out (	OUT_15_POH_CL,	para_s.Out_Val_15_s16);
END_IF

IF para_s.Out_Cfg_16_s16 = PWM_MODE THEN
	out (	OUT_16_POH,	para_s.Out_Val_16_s16);
ELSIF para_s.Out_Cfg_16_s16 = PWM_CURRENT_MODE THEN
	out (	OUT_16_POH_CL,	para_s.Out_Val_16_s16);
END_IF

IF para_s.Out_Cfg_17_s16 = PWM_MODE THEN
	out (	OUT_17_POH,	para_s.Out_Val_17_s16);
ELSIF para_s.Out_Cfg_17_s16 = PWM_CURRENT_MODE THEN
	out (	OUT_17_POH_CL,	para_s.Out_Val_17_s16);
END_IF

IF para_s.Out_Cfg_18_s16 = PWM_MODE THEN
	out (	OUT_18_POH,	para_s.Out_Val_18_s16);
ELSIF para_s.Out_Cfg_18_s16 = PWM_CURRENT_MODE THEN
	out (	OUT_18_POH_CL,	para_s.Out_Val_18_s16);
END_IF
END_ACTION
ACTION out_POL:
(* Proportional output Low side PWM *)

IF para_s.Out_Cfg_37_s16 = PWM_MODE THEN
	out (	OUT_37_POL,	para_s.Out_Val_37_s16);
ELSIF para_s.Out_Cfg_37_s16 = PWM_CURRENT_MODE THEN
	out (	OUT_37_POL_CL,	para_s.Out_Val_37_s16);
END_IF

IF para_s.Out_Cfg_38_s16 = PWM_MODE THEN
	out (	OUT_38_POL,	para_s.Out_Val_38_s16);
ELSIF para_s.Out_Cfg_38_s16 = PWM_CURRENT_MODE THEN
	out (	OUT_38_POL_CL,	para_s.Out_Val_38_s16);
END_IF

IF para_s.Out_Cfg_39_s16 = PWM_MODE THEN
	out (	OUT_39_POL,	para_s.Out_Val_39_s16);
ELSIF para_s.Out_Cfg_39_s16 = PWM_CURRENT_MODE THEN
	out (	OUT_39_POL_CL,	para_s.Out_Val_39_s16);
END_IF

IF para_s.Out_Cfg_40_s16 = PWM_MODE THEN
	out (	OUT_40_POL,	para_s.Out_Val_40_s16);
ELSIF para_s.Out_Cfg_40_s16 = PWM_CURRENT_MODE THEN
	out (	OUT_40_POL_CL,	para_s.Out_Val_40_s16);
END_IF

IF para_s.Out_Cfg_41_s16 = PWM_MODE THEN
	out (	OUT_41_POL,	para_s.Out_Val_14_s16);
ELSIF para_s.Out_Cfg_14_s16 = PWM_CURRENT_MODE THEN
	out (	OUT_41_POL_CL,	para_s.Out_Val_41_s16);
END_IF

IF para_s.Out_Cfg_42_s16 = PWM_MODE THEN
	out (	OUT_42_POL,	para_s.Out_Val_42_s16);
ELSIF para_s.Out_Cfg_42_s16 = PWM_CURRENT_MODE THEN
	out (	OUT_42_POL_CL,	para_s.Out_Val_42_s16);
END_IF

IF para_s.Out_Cfg_43_s16 = PWM_MODE THEN
	out (	OUT_43_POL,	para_s.Out_Val_43_s16);
ELSIF para_s.Out_Cfg_43_s16 = PWM_CURRENT_MODE THEN
	out (	OUT_43_POL_CL,	para_s.Out_Val_43_s16);
END_IF

IF para_s.Out_Cfg_44_s16 = PWM_MODE THEN
	out (	OUT_44_POL,	para_s.Out_Val_44_s16);
ELSIF para_s.Out_Cfg_44_s16 = PWM_CURRENT_MODE THEN
	out (	OUT_44_POL_CL,	para_s.Out_Val_44_s16);
END_IF

IF para_s.Out_Cfg_45_s16 = PWM_MODE THEN
	out (	OUT_45_POL,	para_s.Out_Val_45_s16);
ELSIF para_s.Out_Cfg_45_s16 = PWM_CURRENT_MODE THEN
	out (	OUT_45_POL_CL,	para_s.Out_Val_45_s16);
END_IF

IF para_s.Out_Cfg_46_s16 = PWM_MODE THEN
	out (	OUT_46_POL,	para_s.Out_Val_46_s16);
ELSIF para_s.Out_Cfg_46_s16 = PWM_CURRENT_MODE THEN
	out (	OUT_46_POL_CL,	para_s.Out_Val_46_s16);
END_IF
END_ACTION

(* POU 30_Outputs/out_Current, ST *)
PROGRAM out_Current
VAR
END_VAR
(********************************************************************************)
(***** Получение актуальных значений токов PWM выходов **************************)
(********************************************************************************)

(* Test Code *)
output.iAct_Out_01_ma_s32			:= in( OUT_1_PIC );
output.iAct_Out_02_ma_s32			:= in( OUT_2_PIC );
output.iAct_Out_03_ma_s32			:= in( OUT_3_PIC );
output.iAct_Out_04_ma_s32			:= in( OUT_4_PIC );

(* code for test *)
output.iAct_Out_02_ma_s32			:= in( OUT_2_PIC );
output.iAct_Out_03_ma_s32			:= in( OUT_3_PIC );
output.iAct_Out_04_ma_s32			:= in( OUT_4_PIC );
output.iAct_Out_05_ma_s32			:= in( OUT_5_PIC );

output.iAct_Out_01_ma_s32			:= in( OUT_1_PIC );
output.iAct_Out_02_ma_s32			:= in( OUT_2_PIC );
output.iAct_Out_03_ma_s32			:= in( OUT_3_PIC );
output.iAct_Out_04_ma_s32			:= in( OUT_4_PIC );
output.iAct_Out_05_ma_s32			:= in( OUT_5_PIC );
output.iAct_Out_06_ma_s32			:= in( OUT_6_PIC );
output.iAct_Out_07_ma_s32			:= in( OUT_7_PIC );
output.iAct_Out_08_ma_s32			:= in( OUT_8_PIC );
output.iAct_Out_09_ma_s32			:= in( OUT_9_PIC );
output.iAct_Out_10_ma_s32			:= in( OUT_10_PIC);
output.iAct_Out_11_ma_s32			:= in( OUT_11_PIC);
output.iAct_Out_12_ma_s32			:= in( OUT_12_PIC);
output.iAct_Out_13_ma_s32			:= in( OUT_13_PIC);
output.iAct_Out_14_ma_s32			:= in( OUT_14_PIC);
output.iAct_Out_15_ma_s32			:= in( OUT_15_PIC);
output.iAct_Out_16_ma_s32			:= in( OUT_16_PIC);
output.iAct_Out_17_ma_s32			:= in( OUT_17_PIC);
output.iAct_Out_18_ma_s32			:= in( OUT_18_PIC);
output.iAct_Out_19_ma_s32			:= in( OUT_19_PIC);
output.iAct_Out_20_ma_s32			:= in( OUT_20_PIC);
output.iAct_Out_21_ma_s32			:= in( OUT_21_PIC);
output.iAct_Out_22_ma_s32			:= in( OUT_22_PIC);
output.iAct_Out_23_ma_s32			:= in( OUT_23_PIC);
output.iAct_Out_24_ma_s32			:= in( OUT_24_PIC);
output.iAct_Out_25_ma_s32			:= in( OUT_25_PIC);
output.iAct_Out_26_ma_s32			:= in( OUT_26_PIC);
output.iAct_Out_27_ma_s32			:= in( OUT_27_PIC);
output.iAct_Out_28_ma_s32			:= in( OUT_28_PIC);
output.iAct_Out_29_ma_s32			:= in( OUT_29_PIC);
output.iAct_Out_30_ma_s32			:= in( OUT_30_PIC);
output.iAct_Out_31_ma_s32			:= in( OUT_31_PIC);
output.iAct_Out_32_ma_s32			:= in( OUT_32_PIC);
output.iAct_Out_37_ma_s32			:= in( OUT_37_PIC);
output.iAct_Out_38_ma_s32			:= in( OUT_38_PIC);
output.iAct_Out_39_ma_s32			:= in( OUT_39_PIC);
output.iAct_Out_40_ma_s32			:= in( OUT_40_PIC);
output.iAct_Out_41_ma_s32			:= in( OUT_41_PIC);
output.iAct_Out_42_ma_s32			:= in( OUT_42_PIC);
output.iAct_Out_43_ma_s32			:= in( OUT_43_PIC);
output.iAct_Out_44_ma_s32			:= in( OUT_44_PIC);
output.iAct_Out_45_ma_s32			:= in( OUT_45_PIC);
output.iAct_Out_46_ma_s32			:= in( OUT_46_PIC);
END_PROGRAM

(* POU 30_Outputs/out_Status, ST *)
PROGRAM out_Status
VAR

	out_as: ARRAY [1..75] OF out_ts;	(* Structure with the extended output information *)

END_VAR
out_getStatusxt(OUT_1_POH,		ADR(out_as[1]));
out_getStatusxt(OUT_2_POH,		ADR(out_as[2]));
out_getStatusxt(OUT_3_POH, 	ADR(out_as[3]));
out_getStatusxt(OUT_4_POH, 	ADR(out_as[4]));
out_getStatusxt(OUT_5_POH, 	ADR(out_as[5]));
out_getStatusxt(OUT_6_POH, 	ADR(out_as[6]));
out_getStatusxt(OUT_7_POH, 	ADR(out_as[7]));
out_getStatusxt(OUT_8_POH, 	ADR(out_as[8]));
out_getStatusxt(OUT_9_POH, 	ADR(out_as[9]));
out_getStatusxt(OUT_10_POH, 	ADR(out_as[10]));
out_getStatusxt(OUT_11_POH, 	ADR(out_as[11]));
out_getStatusxt(OUT_12_POH, 	ADR(out_as[12]));
out_getStatusxt(OUT_13_POH, 	ADR(out_as[13]));
out_getStatusxt(OUT_14_POH,	ADR(out_as[14]));
out_getStatusxt(OUT_15_POH,	ADR(out_as[15]));
out_getStatusxt(OUT_16_POH, 	ADR(out_as[16]));
out_getStatusxt(OUT_17_POH,	ADR(out_as[17]));
out_getStatusxt(OUT_18_POH,	ADR(out_as[18]));
out_getStatusxt(OUT_19_DOH,	ADR(out_as[19]));
out_getStatusxt(OUT_20_DOH,	ADR(out_as[20]));
out_getStatusxt(OUT_21_DOH,	ADR(out_as[21]));
out_getStatusxt(OUT_22_DOH,	ADR(out_as[22]));
out_getStatusxt(OUT_23_DOH,	ADR(out_as[23]));
out_getStatusxt(OUT_24_DOH,	ADR(out_as[24]));
out_getStatusxt(OUT_25_DOH,	ADR(out_as[25]));
out_getStatusxt(OUT_26_DOH,	ADR(out_as[26]));
out_getStatusxt(OUT_27_DOH,	ADR(out_as[27]));
out_getStatusxt(OUT_28_DOH,	ADR(out_as[28]));
out_getStatusxt(OUT_29_DOH,	ADR(out_as[29]));
out_getStatusxt(OUT_30_DOH,	ADR(out_as[30]));
out_getStatusxt(OUT_31_DOH,	ADR(out_as[31]));
out_getStatusxt(OUT_32_DOH,	ADR(out_as[32]));
out_getStatusxt(OUT_33_POH,	ADR(out_as[33]));
out_getStatusxt(OUT_34_POH,	ADR(out_as[34]));
out_getStatusxt(OUT_35_POH,	ADR(out_as[35]));
out_getStatusxt(OUT_36_POH,	ADR(out_as[36]));
out_getStatusxt(OUT_37_POL,	ADR(out_as[37]));
out_getStatusxt(OUT_38_POL,	ADR(out_as[38]));
out_getStatusxt(OUT_39_POL,	ADR(out_as[39]));
out_getStatusxt(OUT_40_POL,	ADR(out_as[40]));
out_getStatusxt(OUT_41_POL,	ADR(out_as[41]));
out_getStatusxt(OUT_42_POL,	ADR(out_as[42]));
out_getStatusxt(OUT_43_POL,	ADR(out_as[43]));
out_getStatusxt(OUT_44_POL,	ADR(out_as[44]));
out_getStatusxt(OUT_45_POL,	ADR(out_as[45]));
out_getStatusxt(OUT_46_POL,	ADR(out_as[46]));
out_getStatusxt(OUT_47_AOV,	ADR(out_as[47]));

(* test code *)
out_getStatusxt(OUT_42_POL,	ADR(out_as[42]));
out_getStatusxt(OUT_43_POL,	ADR(out_as[43]));
out_getStatusxt(OUT_44_POL,	ADR(out_as[44]));
out_getStatusxt(OUT_45_POL,	ADR(out_as[45]));
out_getStatusxt(OUT_46_POL,	ADR(out_as[46]));
out_getStatusxt(OUT_47_AOV,	ADR(out_as[47]));
END_PROGRAM

(* POU 60_Error handling/Process Errors/proc_Err_DIG_outs, ST *)
PROGRAM proc_Err_DIG_outs
VAR

END_VAR
;
END_PROGRAM

(* POU 60_Error handling/Process Errors/proc_Err_Inputs, ST *)
PROGRAM proc_Err_Inputs
VAR

(*		Here we process errors from sensors, or HMI - which have to be calibrated at the beginning
		 = 0 no error, > 0 error
		Encoding of error bits:
			Bit 0x0000 = no error
			Bit 0x0004 = potentiometer slider < lower error threshold value (only if error threshold value >0)
			Bit 0x0008 = potentiometer slider > upper error threshold value
			Bit 0x0020 = potentiometer slider > max poti voltage + 5% (e.g. 10,5V for a 10V input and max voltage = nominal voltage 10V). 
		This bit can not be set if the defined max poti voltage is already greater than the ADC input range!    
			Bit 0x0001 = Current through defined current channel out of defined limit (not defined by inext_getPotiStatus(), but set here separetely)
*)
END_VAR
VAR CONSTANT

END_VAR
;
END_PROGRAM

(* POU 60_Error handling/Process Errors/proc_Err_Parameters, ST *)
PROGRAM proc_Err_Parameters
VAR
END_VAR
;
END_PROGRAM

(* POU 60_Error handling/Process Errors/proc_Err_Power, ST *)
PROGRAM proc_Err_Power
VAR
	ProcessErr1_fb: 			handleError;
	ProcessErr2_fb: 			handleError;
	ProcessErr3_fb: 			handleError;
	ProcessErr4_fb: 			handleError;


	uSupplyVB_mV_u16: UINT;
	uSupplyVSS2_mV_u16: UINT;
	uSupplyVSS1_mV_u16: UINT;
END_VAR
uSupplyVB_mV_u16 		:= sys_getSupply( VB );					(* voltage level of VB [mV] *)

(*******************************************************************************************)
(******************** @ERR: 24V too high ****************************************************)
(*******************************************************************************************)
ProcessErr1_fb(
	stErrorCondition_b8	:= stStartlock_b8 AND uSupplyVB_mV_u16 > 32000 ,		(* error condition *)
	stQuitCondition_b8	:= TRUE ,								(* reset condition *)
	tiDelay_u16				:= DELAY_STANDARD,					(* debouncing time [ms] *)
	numErr_code_u16		:= ERR_SUPPLY_VB_HIGH,						(* start at 16#8000 *)
	numErr_nbr_u8			:= 0,								(* error no for B-s text inputs *)
	bSave_b8					:= TRUE,									(* save in EEPROM *)
	tiCycle_s16				:= CYCLE,								(* current cycle time *)
	bFlag_b8					=> Err.Supply_vb_high_b8 );		(* flag induces reaction in _RUN block*)



(*******************************************************************************************)
(******************** @ERR: 24V too low ****************************************************)
(*******************************************************************************************)
ProcessErr2_fb(
	stErrorCondition_b8	:= stStartlock_b8 AND uSupplyVB_mV_u16 < 18000 ,		(* error condition *)
	stQuitCondition_b8	:= TRUE ,								(* reset condition *)
	tiDelay_u16				:= DELAY_STANDARD,					(* debouncing time [ms] *)
	numErr_code_u16		:= ERR_SUPPLY_VB_LOW,						(* start at 16#8000 *)
	numErr_nbr_u8			:= 0,								(* error no for B-s text inputs *)
	bSave_b8					:= TRUE,									(* save in EEPROM *)
	tiCycle_s16				:= CYCLE,								(* current cycle time *)
	bFlag_b8					=> Err.Supply_vb_low_b8 );		(* flag induces reaction in _RUN block*)


(*******************************************************************************************)
(******************** @ERR: VSS1 ***********************************************************)
(*******************************************************************************************)
uSupplyVSS1_mV_u16	:= sys_getSupply( VSS_1 );				(* voltage level of VSS1 [mV] *)

ProcessErr3_fb(
	stErrorCondition_b8	:= stStartlock_b8 AND
									(uSupplyVSS1_mV_u16 < 4500 OR	uSupplyVSS1_mV_u16 > 5500),		(* error condition *)
	stQuitCondition_b8	:= TRUE,									(* reset condition *)
	tiDelay_u16				:= DELAY_STANDARD,					(* debouncing time [ms] *)
	numErr_code_u16		:= ERR_SUPPLY_VSS1,					(* start at 16#8000 *)
	numErr_nbr_u8			:= 0,										(* error no for B-s text inputs *)
	bSave_b8					:= TRUE,									(* save in EEPROM *)
	tiCycle_s16				:= CYCLE,								(* current cycle time *)
	bFlag_b8					=> Err.Supply_vss1_b8 );			(* flag induces reaction in _RUN block*)


(*******************************************************************************************)
(******************** @ERR: VSS2 ***********************************************************)
(*******************************************************************************************)
uSupplyVSS2_mV_u16	:= sys_getSupply( VSS_2 );		(* voltage level of VSS2 [mV] *)

ProcessErr4_fb(
	stErrorCondition_b8	:= stStartlock_b8 AND
									(uSupplyVSS2_mV_u16 < 9500 OR uSupplyVSS2_mV_u16 > 10500),	(* error condition *)
	stQuitCondition_b8	:= TRUE,									(* reset condition *)
	tiDelay_u16				:= DELAY_STANDARD,					(* debouncing time [ms] *)
	numErr_code_u16		:= ERR_SUPPLY_VSS2,					(* start at 16#8000 *)
	numErr_nbr_u8			:= 0,										(* error no for B-s text inputs *)
	bSave_b8					:= TRUE,									(* save in EEPROM *)
	tiCycle_s16				:= CYCLE,								(* current cycle time *)
	bFlag_b8					=> Err.Supply_vss2_b8 );			(* flag induces reaction in _RUN block*)
END_PROGRAM

(* POU 60_Error handling/Process Errors/proc_Err_PWM, ST *)
PROGRAM proc_Err_PWM
VAR
	ProcessErr1_fb: 			handleError;
	ProcessErr2_fb: 			handleError;
	ProcessErr3_fb: 			handleError;
	ProcessErr4_fb: 			handleError;
	ProcessErr5_fb: 			handleError;
	ProcessErr6_fb: 			handleError;
	ProcessErr7_fb: 			handleError;
	ProcessErr8_fb: 			handleError;

	ProcessErr9_fb: 			handleError;
	ProcessErr10_fb: 			handleError;
	ProcessErr11_fb: 			handleError;
	ProcessErr12_fb: 			handleError;



END_VAR
;
END_PROGRAM

(* POU 60_Error handling/Process Errors/proc_Err_Sensors, ST *)
PROGRAM proc_Err_Sensors
VAR
	ProcessErr1_fb				: handleError;

END_VAR
VAR CONSTANT

END_VAR
;
END_PROGRAM

(* POU 60_Error handling/Process Errors/proc_Err_Status, ST *)
PROGRAM proc_Err_Status
VAR
	ProcessErr1_fb		: handleError;


END_VAR
;
END_PROGRAM

(* POU 10_Inputs/Function Blocks/calc_deadband, ST *)
FUNCTION calc_deadband : INT
VAR_INPUT
	iInput:			INT;	(* input setpoint (-1000..1000) *)
	iDeadband:	INT;	(* deadband in % of poti range [0..100] *)
END_VAR
VAR
	tmp:	INT;
END_VAR
iInput := LIMIT(-1000, iInput, 1000);
iDeadband := LIMIT(0, iDeadband, 100);

(* convert from percent *)
iDeadband := iDeadband * 10;

(* calculation of deadband *)
IF iInput > 0 THEN
	tmp := iInput - iDeadband;
	tmp := MAX(tmp, 0);
ELSE
	tmp := iInput + iDeadband;
	tmp := MIN(tmp, 0);
END_IF

calc_deadband := LIMIT( -1000, DINT_TO_INT(INT_TO_DINT(tmp) * 1000 / (1000 - iDeadband)), 1000);
END_FUNCTION

(* POU 05_Basic_Calc/conv_mV_to_dig, ST *)
FUNCTION conv_mV_to_dig : INT
(* Функция конвертации входного напряжения из [0; vMax] в цифровой сигнал  [0; 511] *)
(* Функция возвращает -1, если введены не верные входные параметры *)
VAR_INPUT
	in_mV_s16			: INT;		(* Входной сигнал напряжения, мВ *)
	U_lim_mV_s16		: INT;		(* Максимально допустимое напряжение на входе, мВ *)
END_VAR
VAR
	dig_raw_s16			: INT;		(* Конвертированный сигнал, без округления *)
END_VAR
	(* Проверка на правильность входных данных *)
	IF (in_mV_s16 < 0 OR in_mV_s16 > U_lim_mV_s16) THEN
		(* Входные данные не верные *)
		conv_mV_to_dig := -1;
	ELSE

		(* Конвертация входного сигнала *)
		dig_raw_s16 	:= in_mV_s16 * 5110 / U_lim_mV_s16;

		(* Округление конвертированного сигнала в большую сторону *)
		IF (dig_raw_s16 MOD 10) = 0 THEN
			conv_mV_to_dig := dig_raw_s16/10;
		ELSE
			conv_mV_to_dig := dig_raw_s16/10 + 1;
		END_IF

	END_IF
END_FUNCTION

(* POU 10_Inputs/Function Blocks/Get_PR2_25, ST *)
FUNCTION_BLOCK Get_PR2_25
(* V. Lewitan, DCRU, 08/08-2011, ver 1.0
V. Lewitan, ver 2.0, adapted to RC30, 01/05-2012
*)
VAR_INPUT
	Chn_u32: DWORD;
END_VAR
VAR_OUTPUT
	p0p01bar_s16: INT;
	stPR2_u8: BYTE;
END_VAR
VAR
	v_mV_s16: INT;
END_VAR
v_mV_s16 := DINT_TO_INT( in(Chn_u32));

IF v_mV_s16 < 350 THEN
stPR2_u8 := 2#011;
ELSIF v_mV_s16 > 4650 THEN
stPR2_u8 := 2#101;
ELSE (* no error, fb initialized *)
stPR2_u8 := 2#001;
END_IF

p0p01bar_s16 := Scale_fun_s16( v_mV_s16 , 500, 4500, 0, 2500);
END_FUNCTION_BLOCK

(* POU 05_Basic_Calc/Scale_fun_s16, ST *)
(**********************************************************************************************************
* (c) Copyright by BOSCH REXROTH AG, all rights reserved *
***********************************************************************************************************
PROJECT:   Universal Scale Function
Added 19/01-2011. Weronika Melija,  Bosch Rexroth Russia
Checked 13/05 -2011. Vitaly Lewitan, DCRU/MA-SMC
Short Description
-	Linear Scalling Function 
************************************************************************************************************)
FUNCTION Scale_fun_s16 : INT
VAR_INPUT
	input_s16				:		INT;
	x1_s16					:		INT;
	x2_s16					:		INT;
	y1_s16					:		INT;
	y2_s16					: 		INT;
END_VAR
VAR
	Out_Raw_s16		:		INT;
END_VAR
(* linear scaling *)
IF input_s16 <= x1_s16 THEN
	Out_Raw_s16 := y1_s16;	(* No calculations *)
ELSIF input_s16 >= x2_s16  THEN
	Out_Raw_s16 := y2_s16;	(* No calculations *)
ELSE								(* Calculate Scale Function *)
	Out_Raw_s16 := DINT_TO_INT ( INT_TO_DINT(input_s16 - x1_s16)  *   (y2_s16 - y1_s16)   /   (x2_s16 - x1_s16) + y1_s16);
END_IF
(************************** Limiting *******************************************)
IF y1_s16 <= y2_s16 THEN
	Scale_fun_s16 := LIMIT(y1_s16,  Out_Raw_s16, y2_s16);
ELSIF y1_s16 >  y2_s16 THEN
	Scale_fun_s16 := LIMIT(y2_s16, Out_Raw_s16, y1_s16 );
ELSE
	Scale_fun_s16 := LIMIT(y1_s16,  Out_Raw_s16, y2_s16);
END_IF
(**********************************************************************************)
END_FUNCTION

(* POU 10_Inputs/Function Blocks/Get_PR2_50, ST *)
FUNCTION_BLOCK Get_PR2_50
(* V. Lewitan, DCRU, 08/08-2011, ver 1.0
V. Lewitan, ver 2.0, adapted to RC30, 01/05-2012
*)
VAR_INPUT
	Chn_u32: DWORD;
END_VAR
VAR_OUTPUT
	p0p01bar_s16: INT;
	stPR2_u8: BYTE;
END_VAR
VAR
	v_mV_s16: INT;
END_VAR
v_mV_s16 := DINT_TO_INT( in(Chn_u32));

IF v_mV_s16 < 350 THEN
stPR2_u8 := 2#011;
ELSIF v_mV_s16 > 4650 THEN
stPR2_u8 := 2#101;
ELSE (* no error, fb initialized *)
stPR2_u8 := 2#001;
END_IF

p0p01bar_s16 := Scale_fun_s16( v_mV_s16 , 500, 4500, 0, 5000);
END_FUNCTION_BLOCK

(* POU 10_Inputs/Function Blocks/Get_PR2_600, ST *)
FUNCTION_BLOCK Get_PR2_600
(* V. Lewitan, DCRU, 08/08-2011, ver 1.0
V. Lewitan, ver 2.0, adapted to RC30, 01/05-2012
*)
VAR_INPUT
	Chn_u32: DWORD;
END_VAR
VAR_OUTPUT
	p0p1bar_s16: INT;
	stPR2_u8: BYTE;
END_VAR
VAR
	v_mV_s16: INT;
END_VAR
v_mV_s16 := DINT_TO_INT( in(Chn_u32));

IF v_mV_s16 < 350 THEN
stPR2_u8 := 2#011;
ELSIF v_mV_s16 > 4650 THEN
stPR2_u8 := 2#101;
ELSE (* no error, fb initialized *)
stPR2_u8 := 2#001;
END_IF

p0p1bar_s16 := Scale_fun_s16( v_mV_s16 , 500, 4500, 0, 6000);
END_FUNCTION_BLOCK

(* POU 10_Inputs/Function Blocks/Get_Suction_Pressure, ST *)
FUNCTION_BLOCK Get_Suction_Pressure
(* V. Lewitan, DCRU, 12/01-2013, ver 1.0
V. Lewitan, ver 2.0, adapted to RC30, 01/05-2012
*)
VAR_INPUT
	Chn_u32: DWORD;
END_VAR
VAR_OUTPUT
	p_mbar_s16: INT;
	stPrSen_u8: BYTE;
END_VAR
VAR
	i_uA_s16: INT;
END_VAR
i_uA_s16 := DINT_TO_INT( in(Chn_u32));

IF i_uA_s16 < 1000 THEN
	stPrSen_u8 := 2#011;
ELSIF i_uA_s16 > 20400 THEN
	stPrSen_u8 := 2#101;
ELSE (* no error, fb initialized *)
	stPrSen_u8 := 2#001;
END_IF

p_mbar_s16 := Scale_fun_s16( i_uA_s16 , 0, 20000, -1000, 6000);
END_FUNCTION_BLOCK

(* POU 05_Basic_Calc/eeprom_operations/getEEP_Index, ST *)
(* Функция получает номер ячейки относительно начала текущей страницы *)
FUNCTION getEEP_Index : INT
VAR_INPUT
	EEP_num					: INT;
END_VAR
VAR
	EEP_ELEMENT_OF_PAGE	: INT		:= 256;
END_VAR
getEEP_Index := EEP_num - (EEP_num / EEP_ELEMENT_OF_PAGE) * EEP_ELEMENT_OF_PAGE;
END_FUNCTION

(* POU 05_Basic_Calc/eeprom_operations/getEEP_P3, ST *)
FUNCTION getEEP_P3 : INT
VAR_INPUT
	EEP_num				: INT;
END_VAR
VAR
	EEP_PAGE3_OFFSET	: INT		:= 768;
END_VAR
getEEP_P3	:= EEP_num - EEP_PAGE3_OFFSET;
END_FUNCTION

(* POU 05_Basic_Calc/eeprom_operations/getEEP_Page, ST *)
(* Определение номера страницы eeprom по индексу параметра *)
FUNCTION getEEP_Page : INT
VAR_INPUT
	EEP_num					: INT;
END_VAR
VAR
	EEP_ELEMENT_OF_PAGE	: INT		:= 256;
END_VAR
getEEP_Page := EEP_num / EEP_ELEMENT_OF_PAGE;
END_FUNCTION

(* POU 10_Inputs/Function Blocks/getPedal_Sensor_fb, ST *)
(*************************************************************************************
* FUNCTION BLOCK: in_pedal_or_sensor
*/
* Getting poti calibration parameters, set error intervals and getting poti calibrated
	value [-1000, 1000 ], taking into account deadband
*
*	\param[in]
*	\param[in/out]
*	\param[out]
*
**************************************************************************************
* (c) Copyright by BOSCH REXROTH AG, all rights reserved *
**************************************************************************************
*
* PROJECT:	
* VERSION INFORMATION: 
*
* REVISION HISTORY:
*
*	V1.00, Vitaly Lewitan, DCRU-MA/SMC
*	23.03.2012 - Basic Version
*
*************************************************************************************)

FUNCTION_BLOCK getPedal_Sensor_fb
VAR_OUTPUT
	poti_s16		:	INT	;	(*	[0 .. 1000]			 Analog poti value of the speed potentiometer	*)
END_VAR
VAR
	poti_min_s16: INT;
	poti_max_s16: INT;
	poti_emin_s16: INT;
	poti_emax_s16: INT;
	poti_raw_s16: INT;
END_VAR

VAR_INPUT
	PotiAdjust_s16: INT;
	PotiChannel_u32: DWORD;
	DeadBand_s16: INT;
END_VAR
(* get poti adjustment values *)
poti_min_s16 := inext_getPotiMin( PotiAdjust_s16 );
poti_max_s16 := LIMIT(501, inext_getPotiMax( PotiAdjust_s16 ), 1000);

(*derive error thresholds from adjustment values *)
IF poti_min_s16 >= 50 THEN
	poti_emin_s16 := poti_min_s16 - 50;
ELSE
	poti_emin_s16 := 0;
END_IF

